C01807=1039.398,-71.584,-77.475,168.803,36.714,156.907
C01808=1039.391,-71.834,-77.463,168.801,36.714,156.907
C01809=1039.386,-72.084,-77.451,168.798,36.713,156.907
C01810=1039.380,-72.333,-77.439,168.796,36.713,156.907
C01811=1039.374,-72.584,-77.428,168.793,36.713,156.907
C01812=1039.368,-72.833,-77.417,168.791,36.713,156.907
C01813=1039.361,-73.083,-77.405,168.789,36.713,156.907
C01814=1039.356,-73.332,-77.394,168.786,36.713,156.907
C01815=1039.349,-73.582,-77.382,168.784,36.713,156.907
C01816=1039.344,-73.832,-77.371,168.781,36.713,156.907
C01817=1039.337,-74.082,-77.360,168.779,36.713,156.907
C01818=1039.331,-74.331,-77.348,168.776,36.713,156.907
C01819=1039.325,-74.581,-77.337,168.774,36.713,156.907
C01820=1039.319,-74.831,-77.325,168.772,36.713,156.907
C01821=1039.313,-75.080,-77.314,168.769,36.713,156.907
C01822=1039.306,-75.330,-77.303,168.767,36.713,156.907
C01823=1039.301,-75.580,-77.292,168.764,36.713,156.907
C01824=1039.294,-75.829,-77.280,168.762,36.713,156.907
C01825=1039.288,-76.079,-77.269,168.759,36.713,156.907
C01826=1039.282,-76.329,-77.258,168.757,36.713,156.907
C01827=1039.276,-76.578,-77.246,168.754,36.713,156.907
C01828=1039.269,-76.828,-77.235,168.752,36.714,156.907
C01829=1039.264,-77.077,-77.224,168.749,36.714,156.907
C01830=1039.257,-77.328,-77.213,168.747,36.714,156.907
C01831=1039.251,-77.576,-77.201,168.745,36.714,156.907
C01832=1039.244,-77.826,-77.190,168.742,36.714,156.907
C01833=1039.238,-78.076,-77.180,168.740,36.714,156.907
C01834=1039.232,-78.326,-77.168,168.737,36.714,156.907
C01835=1039.226,-78.575,-77.157,168.735,36.714,156.907
C01836=1039.220,-78.825,-77.146,168.732,36.714,156.907
C01837=1039.214,-79.075,-77.135,168.730,36.714,156.907
C01838=1039.208,-79.325,-77.123,168.727,36.714,156.907
C01839=1039.202,-79.574,-77.113,168.725,36.714,156.907
C01840=1039.196,-79.824,-77.101,168.722,36.714,156.907
C01841=1039.190,-80.074,-77.090,168.720,36.714,156.907
C01842=1039.182,-80.323,-77.079,168.717,36.714,156.907
C01843=1039.177,-80.573,-77.068,168.715,36.714,156.907
C01844=1039.170,-80.823,-77.057,168.712,36.714,156.907
C01845=1039.164,-81.072,-77.047,168.710,36.714,156.907
C01846=1039.158,-81.321,-77.036,168.707,36.715,156.907
C01847=1039.152,-81.572,-77.025,168.705,36.715,156.907
C01848=1039.145,-81.821,-77.014,168.702,36.715,156.907
C01849=1039.139,-82.071,-77.003,168.700,36.715,156.907
C01850=1039.133,-82.321,-76.992,168.697,36.716,156.908
C01851=1039.126,-82.570,-76.981,168.695,36.716,156.908
C01852=1039.120,-82.820,-76.971,168.692,36.716,156.908
C01853=1039.114,-83.070,-76.959,168.690,36.716,156.908
C01854=1039.108,-83.319,-76.949,168.687,36.716,156.908
C01855=1039.101,-83.605,-76.936,168.684,36.716,156.908
C01856=1039.094,-83.889,-76.924,168.682,36.717,156.908
C01857=1039.087,-84.174,-76.911,168.679,36.717,156.908
C01858=1039.080,-84.459,-76.899,168.676,36.717,156.908
C01859=1039.073,-84.709,-76.889,168.673,36.717,156.908
C01860=1039.067,-84.958,-76.878,168.672,36.718,156.908
C01861=1039.061,-85.209,-76.867,168.669,36.718,156.908
C01862=1039.054,-85.458,-76.856,168.667,36.718,156.908
C01863=1039.049,-85.707,-76.845,168.664,36.718,156.908
C01864=1039.042,-85.957,-76.834,168.662,36.719,156.908
C01865=1039.036,-86.207,-76.825,168.659,36.719,156.908
C01866=1039.030,-86.457,-76.814,168.657,36.719,156.908
C01867=1039.024,-86.707,-76.802,168.654,36.719,156.908
C01868=1039.018,-86.956,-76.792,168.652,36.719,156.908
C01869=1039.012,-87.206,-76.781,168.649,36.719,156.908
C01870=1039.005,-87.456,-76.770,168.647,36.719,156.908
C01871=1038.999,-87.705,-76.760,168.644,36.720,156.908
C01872=1038.993,-87.954,-76.749,168.642,36.720,156.908
C01873=1038.986,-88.205,-76.739,168.639,36.720,156.908
C01874=1038.981,-88.454,-76.728,168.637,36.721,156.908
C01875=1038.975,-88.704,-76.717,168.634,36.721,156.908
C01876=1038.968,-88.954,-76.707,168.631,36.721,156.908
C01877=1038.962,-89.203,-76.696,168.629,36.721,156.908
C01878=1038.957,-89.453,-76.685,168.626,36.721,156.908
C01879=1038.950,-89.703,-76.675,168.624,36.721,156.908
C01880=1038.944,-89.953,-76.664,168.621,36.722,156.908
C01881=1038.937,-90.202,-76.654,168.619,36.722,156.908
C01882=1038.932,-90.451,-76.643,168.616,36.722,156.908
C01883=1038.926,-90.702,-76.632,168.614,36.723,156.909
C01884=1038.919,-90.951,-76.622,168.611,36.723,156.909
C01885=1038.913,-91.201,-76.611,168.609,36.723,156.909
C01886=1038.907,-91.450,-76.601,168.606,36.723,156.909
C01887=1038.902,-91.700,-76.591,168.604,36.723,156.909
C01888=1038.895,-91.950,-76.579,168.601,36.724,156.909
C01889=1038.889,-92.200,-76.569,168.599,36.724,156.909
C01890=1038.883,-92.450,-76.559,168.596,36.724,156.909
C01891=1038.877,-92.699,-76.549,168.593,36.725,156.909
C01892=1038.870,-92.949,-76.537,168.591,36.725,156.909
C01893=1038.864,-93.199,-76.528,168.588,36.725,156.909
C01894=1038.859,-93.448,-76.517,168.586,36.726,156.909
C01895=1038.853,-93.698,-76.506,168.583,36.726,156.909
C01896=1038.847,-93.948,-76.497,168.581,36.726,156.909
C01897=1038.841,-94.197,-76.486,168.578,36.726,156.909
C01898=1038.834,-94.447,-76.475,168.576,36.726,156.909
C01899=1038.828,-94.697,-76.465,168.573,36.727,156.909
C01900=1038.823,-94.947,-76.454,168.571,36.727,156.909
C01901=1038.816,-95.196,-76.444,168.568,36.727,156.909
C01902=1038.811,-95.446,-76.434,168.566,36.728,156.909
C01903=1038.804,-95.695,-76.423,168.563,36.728,156.909
C01904=1038.799,-95.945,-76.413,168.561,36.728,156.909
C01905=1038.792,-96.195,-76.402,168.559,36.728,156.909
C01906=1038.786,-96.445,-76.392,168.556,36.728,156.909
C01907=1038.780,-96.694,-76.382,168.554,36.729,156.909
C01908=1038.774,-96.944,-76.372,168.551,36.729,156.909
C01909=1038.769,-97.194,-76.361,168.549,36.730,156.910
C01910=1038.762,-97.443,-76.351,168.546,36.730,156.910
C01911=1038.756,-97.693,-76.341,168.544,36.730,156.910
C01912=1038.751,-97.943,-76.331,168.541,36.730,156.910
C01913=1038.744,-98.193,-76.320,168.538,36.731,156.910
C01914=1038.737,-98.443,-76.311,168.536,36.731,156.910
C01915=1038.732,-98.692,-76.300,168.533,36.732,156.910
C01916=1038.725,-98.942,-76.290,168.531,36.732,156.910
C01917=1038.719,-99.191,-76.280,168.528,36.732,156.910
C01918=1038.714,-99.441,-76.270,168.525,36.733,156.910
C01919=1038.706,-99.729,-76.259,168.522,36.734,156.910
C01920=1038.699,-100.015,-76.247,168.519,36.734,156.910
C01921=1038.692,-100.303,-76.235,168.517,36.734,156.910
C01922=1038.685,-100.590,-76.224,168.514,36.735,156.910
C01923=1038.679,-100.840,-76.214,168.511,36.735,156.910
C01924=1038.673,-101.089,-76.203,168.508,36.736,156.911
C01925=1038.667,-101.339,-76.194,168.506,36.737,156.911
C01926=1038.660,-101.589,-76.184,168.503,36.737,156.911
C01927=1038.655,-101.839,-76.173,168.501,36.737,156.911
C01928=1038.649,-102.088,-76.164,168.498,36.737,156.911
C01929=1038.642,-102.338,-76.154,168.495,36.738,156.911
C01930=1038.636,-102.587,-76.144,168.494,36.739,156.911
C01931=1038.630,-102.837,-76.134,168.491,36.739,156.911
C01932=1038.624,-103.087,-76.124,168.489,36.739,156.911
C01933=1038.618,-103.336,-76.114,168.486,36.740,156.911
C01934=1038.612,-103.587,-76.104,168.483,36.740,156.911
C01935=1038.606,-103.836,-76.094,168.481,36.741,156.911
C01936=1038.600,-104.086,-76.084,168.478,36.741,156.911
C01937=1038.594,-104.335,-76.074,168.476,36.741,156.911
C01938=1038.588,-104.585,-76.064,168.473,36.742,156.911
C01939=1038.582,-104.835,-76.054,168.470,36.743,156.912
C01940=1038.576,-105.085,-76.045,168.468,36.743,156.912
C01941=1038.570,-105.335,-76.035,168.465,36.743,156.912
C01942=1038.564,-105.584,-76.024,168.463,36.744,156.912
C01943=1038.558,-105.834,-76.015,168.460,36.745,156.912
C01944=1038.552,-106.084,-76.005,168.457,36.745,156.912
C01945=1038.545,-106.334,-75.996,168.455,36.745,156.912
C01946=1038.539,-106.583,-75.986,168.452,36.746,156.912
C01947=1038.533,-106.833,-75.975,168.449,36.747,156.912
C01948=1038.527,-107.083,-75.966,168.447,36.747,156.912
///RCONF 1,0,0,0,1,0,0,0,0,0,0,0,0,0,0,0,0,0,0,0,0,0,0,0
C01949=1038.521,-107.333,-75.956,168.444,36.747,156.912
C01950=1038.515,-107.582,-75.947,168.442,36.748,156.912
C01951=1038.509,-107.832,-75.937,168.440,36.749,156.913
C01952=1038.503,-108.082,-75.927,168.437,36.749,156.913
C01953=1038.496,-108.332,-75.918,168.435,36.749,156.913
C01954=1038.490,-108.582,-75.908,168.432,36.750,156.913
C01955=1038.484,-108.831,-75.899,168.429,36.751,156.913
C01956=1038.479,-109.081,-75.889,168.427,36.751,156.913
C01957=1038.473,-109.331,-75.879,168.424,36.752,156.913
C01958=1038.467,-109.580,-75.870,168.422,36.753,156.913
C01959=1038.461,-109.830,-75.860,168.419,36.753,156.913
C01960=1038.454,-110.079,-75.850,168.416,36.754,156.913
C01961=1038.448,-110.329,-75.840,168.414,36.754,156.913
C01962=1038.442,-110.579,-75.831,168.411,36.755,156.914
C01963=1038.436,-110.829,-75.821,168.408,36.756,156.914
C01964=1038.430,-111.079,-75.812,168.406,36.756,156.914
C01965=1038.424,-111.329,-75.803,168.403,36.757,156.914
C01966=1038.418,-111.579,-75.793,168.400,36.757,156.914
C01967=1038.412,-111.828,-75.784,168.398,36.758,156.914
C01968=1038.406,-112.078,-75.774,168.395,36.758,156.914
C01969=1038.400,-112.327,-75.765,168.393,36.759,156.914
C01970=1038.393,-112.577,-75.755,168.391,36.760,156.914
C01971=1038.387,-112.827,-75.746,168.388,36.760,156.914
C01972=1038.381,-113.077,-75.736,168.386,36.761,156.914
C01973=1038.376,-113.326,-75.727,168.383,36.762,156.915
C01974=1038.369,-113.576,-75.717,168.380,36.762,156.915
C01975=1038.363,-113.826,-75.708,168.378,36.762,156.915
C01976=1038.358,-114.076,-75.698,168.375,36.763,156.915
C01977=1038.352,-114.325,-75.688,168.372,36.764,156.915
C01978=1038.345,-114.576,-75.680,168.370,36.764,156.915
C01979=1038.339,-114.825,-75.671,168.367,36.765,156.915
C01980=1038.333,-115.074,-75.661,168.364,36.766,156.915
C01981=1038.327,-115.324,-75.652,168.362,36.766,156.915
C01982=1038.321,-115.574,-75.642,168.359,36.767,156.915
C01983=1038.314,-115.861,-75.631,168.356,36.768,156.916
C01984=1038.307,-116.147,-75.621,168.354,36.769,156.916
C01985=1038.301,-116.433,-75.610,168.351,36.770,156.916
C01986=1038.294,-116.719,-75.599,168.348,36.770,156.916
C01987=1038.288,-116.969,-75.590,168.345,36.771,156.916
C01988=1038.282,-117.219,-75.580,168.342,36.772,156.916
C01989=1038.275,-117.469,-75.572,168.340,36.772,156.916
C01990=1038.269,-117.718,-75.563,168.337,36.773,156.916
C01991=1038.263,-117.968,-75.553,168.334,36.774,156.917
C01992=1038.257,-118.218,-75.544,168.332,36.774,156.917
C01993=1038.251,-118.468,-75.535,168.329,36.775,156.917
C01994=1038.246,-118.717,-75.526,168.326,36.776,156.917
C01995=1038.239,-118.967,-75.516,168.324,36.777,156.917
C01996=1038.233,-119.217,-75.508,168.321,36.777,156.917
C01997=1038.227,-119.467,-75.498,168.319,36.779,156.917
C01998=1038.221,-119.716,-75.489,168.317,36.779,156.917
C01999=1038.215,-119.967,-75.480,168.314,36.780,156.917
C02000=1038.209,-120.216,-75.471,168.311,36.781,156.918
C02001=1038.203,-120.465,-75.461,168.309,36.781,156.918
C02002=1038.197,-120.716,-75.453,168.306,36.782,156.918
C02003=1038.191,-120.965,-75.444,168.303,36.783,156.918
C02004=1038.185,-121.216,-75.435,168.301,36.783,156.918
C02005=1038.179,-121.465,-75.426,168.298,36.784,156.918
C02006=1038.173,-121.715,-75.416,168.295,36.785,156.918
C02007=1038.167,-121.965,-75.407,168.293,36.786,156.918
C02008=1038.161,-122.214,-75.399,168.290,36.787,156.919
C02009=1038.155,-122.464,-75.390,168.287,36.787,156.919
C02010=1038.149,-122.714,-75.380,168.286,36.788,156.919
C02011=1038.143,-122.963,-75.371,168.283,36.789,156.919
C02012=1038.137,-123.213,-75.363,168.280,36.789,156.919
C02013=1038.131,-123.463,-75.353,168.277,36.791,156.919
C02014=1038.125,-123.713,-75.345,168.275,36.791,156.919
C02015=1038.119,-123.963,-75.335,168.272,36.792,156.919
C02016=1038.114,-124.212,-75.327,168.269,36.793,156.920
C02017=1038.107,-124.462,-75.318,168.267,36.793,156.920
C02018=1038.101,-124.712,-75.309,168.264,36.794,156.920
C02019=1038.095,-124.961,-75.300,168.261,36.795,156.920
C02020=1038.089,-125.211,-75.291,168.259,36.796,156.920
C02021=1038.083,-125.461,-75.282,168.256,36.797,156.920
C02022=1038.077,-125.711,-75.273,168.254,36.798,156.920
C02023=1038.071,-125.961,-75.265,168.251,36.799,156.920
C02024=1038.065,-126.210,-75.256,168.249,36.800,156.921
C02025=1038.059,-126.461,-75.247,168.246,36.800,156.921
C02026=1038.053,-126.710,-75.238,168.243,36.802,156.921
C02027=1038.047,-126.960,-75.230,168.241,36.802,156.921
C02028=1038.041,-127.210,-75.221,168.238,36.803,156.921
C02029=1038.035,-127.459,-75.212,168.235,36.804,156.921
C02030=1038.029,-127.709,-75.203,168.233,36.805,156.921
C02031=1038.024,-127.958,-75.194,168.230,36.806,156.922
C02032=1038.019,-128.208,-75.184,168.227,36.806,156.922
C02033=1038.014,-128.458,-75.175,168.225,36.806,156.922
C02034=1038.011,-128.708,-75.164,168.223,36.805,156.921
C02035=1038.008,-128.958,-75.153,168.221,36.804,156.921
C02036=1038.007,-129.208,-75.140,168.219,36.802,156.921
C02037=1038.005,-129.458,-75.128,168.217,36.800,156.921
C02038=1038.005,-129.707,-75.115,168.215,36.798,156.920
C02039=1038.005,-129.957,-75.101,168.213,36.794,156.920
C02040=1038.006,-130.208,-75.086,168.212,36.791,156.919
C02041=1038.009,-130.458,-75.071,168.210,36.787,156.918
C02042=1038.012,-130.707,-75.057,168.209,36.783,156.918
C02043=1038.015,-130.959,-75.041,168.207,36.779,156.917
C02044=1038.019,-131.208,-75.024,168.207,36.773,156.916
C02045=1038.024,-131.459,-75.006,168.205,36.767,156.915
C02046=1038.030,-131.708,-74.989,168.205,36.761,156.914
C02047=1037.689,-131.732,-75.257,168.156,36.967,156.948
C02048=1037.683,-131.483,-75.275,168.158,36.973,156.949
C02049=1037.679,-131.233,-75.293,168.158,36.978,156.950
C02050=1037.674,-130.983,-75.309,168.160,36.984,156.951
C02051=1037.671,-130.732,-75.326,168.161,36.988,156.952
C02052=1037.668,-130.483,-75.340,168.162,36.993,156.953
C02053=1037.666,-130.232,-75.356,168.164,36.997,156.954
C02054=1037.665,-129.982,-75.370,168.166,37.000,156.954
C02055=1037.664,-129.732,-75.384,168.167,37.003,156.955
C02056=1037.665,-129.482,-75.397,168.169,37.006,156.955
C02057=1037.665,-129.232,-75.410,168.171,37.007,156.955
C02058=1037.668,-128.983,-75.421,168.173,37.009,156.956
C02059=1037.670,-128.733,-75.433,168.175,37.010,156.956
C02060=1037.674,-128.483,-75.444,168.178,37.011,156.956
C02061=1037.677,-128.232,-75.454,168.180,37.011,156.956
C02062=1037.682,-127.983,-75.464,168.182,37.011,156.956
C02063=1037.688,-127.734,-75.473,168.185,37.010,156.956
C02064=1037.694,-127.484,-75.481,168.188,37.009,156.956
C02065=1037.700,-127.234,-75.490,168.190,37.009,156.956
C02066=1037.706,-126.984,-75.499,168.193,37.007,156.955
C02067=1037.712,-126.735,-75.507,168.196,37.007,156.955
C02068=1037.718,-126.485,-75.516,168.199,37.006,156.955
C02069=1037.724,-126.234,-75.525,168.200,37.004,156.955
C02070=1037.730,-125.986,-75.534,168.203,37.004,156.955
C02071=1037.736,-125.735,-75.543,168.206,37.003,156.955
C02072=1037.741,-125.486,-75.551,168.209,37.002,156.955
C02073=1037.748,-125.236,-75.560,168.211,37.001,156.954
C02074=1037.754,-124.986,-75.569,168.214,37.000,156.954
C02075=1037.760,-124.737,-75.578,168.217,37.000,156.954
C02076=1037.766,-124.486,-75.587,168.219,36.998,156.954
C02077=1037.772,-124.237,-75.596,168.222,36.998,156.954
C02078=1037.778,-123.987,-75.605,168.225,36.997,156.954
C02079=1037.784,-123.737,-75.614,168.228,36.996,156.954
C02080=1037.790,-123.488,-75.622,168.229,36.995,156.953
C02081=1037.796,-123.238,-75.632,168.232,36.994,156.953
C02082=1037.802,-122.987,-75.640,168.235,36.993,156.953
C02083=1037.808,-122.738,-75.650,168.237,36.993,156.953
C02084=1037.814,-122.488,-75.658,168.240,36.992,156.953
C02085=1037.820,-122.238,-75.668,168.243,36.991,156.953
C02086=1037.826,-121.989,-75.676,168.245,36.990,156.953
C02087=1037.832,-121.739,-75.686,168.248,36.989,156.953
C02088=1037.838,-121.489,-75.695,168.251,36.989,156.953
C02089=1037.844,-121.240,-75.703,168.254,36.988,156.952
C02090=1037.850,-120.990,-75.713,168.256,36.987,156.952
C02091=1037.856,-120.740,-75.721,168.258,36.986,156.952
C02092=1037.861,-120.490,-75.731,168.261,36.985,156.952
C02093=1037.868,-120.241,-75.740,168.263,36.984,156.952
C02094=1037.874,-119.990,-75.749,168.266,36.984,156.952
C02095=1037.880,-119.741,-75.758,168.269,36.983,156.952
C02096=1037.886,-119.492,-75.767,168.271,36.982,156.952
C02097=1037.892,-119.241,-75.776,168.274,36.982,156.952
C02098=1037.898,-118.991,-75.786,168.277,36.980,156.951
C02099=1037.904,-118.742,-75.795,168.280,36.980,156.951
C02100=1037.909,-118.492,-75.804,168.282,36.979,156.951
C02101=1037.916,-118.242,-75.813,168.285,36.978,156.951
C02102=1037.923,-117.993,-75.822,168.288,36.978,156.951
C02103=1037.928,-117.744,-75.831,168.290,36.977,156.951
C02104=1037.934,-117.493,-75.840,168.292,36.976,156.951
C02105=1037.940,-117.243,-75.850,168.295,36.975,156.951
C02106=1037.946,-116.994,-75.859,168.297,36.975,156.950
C02107=1037.952,-116.744,-75.868,168.300,36.974,156.950
C02108=1037.959,-116.458,-75.879,168.303,36.973,156.950
C02109=1037.966,-116.172,-75.890,168.306,36.972,156.950
C02110=1037.973,-115.885,-75.901,168.309,36.971,156.950
C02111=1037.980,-115.599,-75.911,168.312,36.971,156.950
C02112=1037.986,-115.349,-75.920,168.315,36.970,156.950
C02113=1037.992,-115.099,-75.929,168.318,36.969,156.950
C02114=1037.998,-114.849,-75.939,168.320,36.969,156.950
C02115=1038.004,-114.600,-75.948,168.323,36.968,156.949
C02116=1038.010,-114.350,-75.958,168.326,36.967,156.949
C02117=1038.016,-114.100,-75.967,168.327,36.967,156.949
C02118=1038.022,-113.851,-75.976,168.330,36.966,156.949
C02119=1038.028,-113.600,-75.985,168.333,36.965,156.949
C02120=1038.034,-113.351,-75.995,168.335,36.964,156.949
C02121=1038.040,-113.101,-76.004,168.338,36.964,156.949
C02122=1038.046,-112.851,-76.014,168.341,36.963,156.949
C02123=1038.052,-112.601,-76.024,168.343,36.962,156.949
C02124=1038.058,-112.352,-76.033,168.346,36.962,156.948
C02125=1038.064,-112.102,-76.042,168.349,36.961,156.948
C02126=1038.070,-111.853,-76.052,168.351,36.960,156.948
C02127=1038.077,-111.603,-76.061,168.354,36.960,156.948
C02128=1038.083,-111.353,-76.071,168.357,36.959,156.948
C02129=1038.089,-111.103,-76.081,168.359,36.958,156.948
C02130=1038.095,-110.853,-76.090,168.362,36.958,156.948
C02131=1038.101,-110.604,-76.100,168.365,36.957,156.948
C02132=1038.106,-110.354,-76.110,168.366,36.957,156.948
C02133=1038.112,-110.104,-76.119,168.369,36.956,156.948
C02134=1038.118,-109.855,-76.129,168.372,36.955,156.948
C02135=1038.125,-109.605,-76.138,168.374,36.955,156.947
C02136=1038.131,-109.355,-76.148,168.377,36.954,156.947
C02137=1038.137,-109.105,-76.157,168.380,36.953,156.947
C02138=1038.143,-108.855,-76.167,168.382,36.953,156.947
C02139=1038.149,-108.606,-76.176,168.385,36.952,156.947
C02140=1038.155,-108.356,-76.186,168.388,36.952,156.947
C02141=1038.162,-108.106,-76.196,168.390,36.951,156.947
C02142=1038.168,-107.856,-76.205,168.393,36.951,156.947
C02143=1038.174,-107.606,-76.215,168.396,36.950,156.947
C02144=1038.180,-107.357,-76.224,168.398,36.949,156.947
C02145=1038.185,-107.107,-76.234,168.401,36.949,156.947
C02146=1038.191,-106.858,-76.244,168.403,36.948,156.947
C02147=1038.198,-106.608,-76.254,168.406,36.948,156.946
C02148=1038.204,-106.358,-76.264,168.409,36.947,156.946
C02149=1038.210,-106.109,-76.273,168.410,36.946,156.946
C02150=1038.215,-105.858,-76.283,168.413,36.946,156.946
C02151=1038.222,-105.609,-76.293,168.416,36.946,156.946
C02152=1038.228,-105.360,-76.303,168.418,36.945,156.946
///RCONF 1,0,0,0,0,0,0,0,0,0,0,0,0,0,0,0,0,0,0,0,0,0,0,0
C02153=1038.234,-105.110,-76.313,168.421,36.944,156.946
C02154=1038.240,-104.860,-76.323,168.423,36.944,156.946
C02155=1038.246,-104.610,-76.332,168.426,36.944,156.946
C02156=1038.252,-104.360,-76.342,168.429,36.943,156.946
C02157=1038.258,-104.111,-76.352,168.431,36.942,156.946
C02158=1038.264,-103.861,-76.362,168.434,36.942,156.946
C02159=1038.270,-103.611,-76.372,168.437,36.942,156.945
C02160=1038.276,-103.361,-76.382,168.439,36.941,156.945
C02161=1038.283,-103.112,-76.392,168.442,36.940,156.945
C02162=1038.288,-102.862,-76.402,168.444,36.940,156.945
C02163=1038.294,-102.612,-76.412,168.447,36.939,156.945
C02164=1038.301,-102.363,-76.422,168.450,36.939,156.945
C02165=1038.307,-102.113,-76.431,168.452,36.939,156.945
C02166=1038.312,-101.863,-76.442,168.455,36.938,156.945
C02167=1038.319,-101.614,-76.452,168.457,36.937,156.945
C02168=1038.325,-101.364,-76.461,168.460,36.937,156.945
C02169=1038.331,-101.114,-76.472,168.462,36.937,156.945
C02170=1038.338,-100.864,-76.482,168.464,36.936,156.945
C02171=1038.344,-100.614,-76.492,168.467,36.936,156.945
C02172=1038.350,-100.327,-76.503,168.470,36.935,156.945
C02173=1038.357,-100.040,-76.515,168.473,36.935,156.944
C02174=1038.365,-99.753,-76.526,168.476,36.934,156.944
C02175=1038.371,-99.466,-76.538,168.479,36.933,156.944
C02176=1038.377,-99.216,-76.548,168.482,36.933,156.944
C02177=1038.384,-98.967,-76.558,168.484,36.932,156.944
C02178=1038.389,-98.717,-76.568,168.487,36.932,156.944
C02179=1038.396,-98.466,-76.578,168.489,36.932,156.944
C02180=1038.403,-98.217,-76.589,168.492,36.931,156.944
C02181=1038.409,-97.967,-76.598,168.495,36.931,156.944
C02182=1038.414,-97.718,-76.609,168.497,36.930,156.944
C02183=1038.421,-97.468,-76.619,168.500,36.930,156.944
C02184=1038.426,-97.218,-76.629,168.502,36.930,156.944
C02185=1038.433,-96.968,-76.639,168.505,36.929,156.944
C02186=1038.438,-96.719,-76.650,168.507,36.929,156.944
C02187=1038.444,-96.469,-76.659,168.510,36.928,156.944
C02188=1038.451,-96.219,-76.671,168.513,36.928,156.944
C02189=1038.457,-95.970,-76.681,168.515,36.928,156.944
C02190=1038.463,-95.720,-76.691,168.518,36.927,156.943
C02191=1038.468,-95.470,-76.702,168.520,36.927,156.943
C02192=1038.475,-95.220,-76.712,168.523,36.927,156.943
C02193=1038.480,-94.971,-76.722,168.525,36.927,156.943
C02194=1038.487,-94.721,-76.732,168.527,36.926,156.943
C02195=1038.493,-94.471,-76.743,168.530,36.926,156.943
C02196=1038.499,-94.222,-76.754,168.532,36.925,156.943
C02197=1038.505,-93.972,-76.764,168.535,36.925,156.943
C02198=1038.511,-93.722,-76.775,168.537,36.925,156.943
C02199=1038.517,-93.473,-76.785,168.540,36.925,156.943
C02200=1038.522,-93.223,-76.795,168.542,36.925,156.943
C02201=1038.530,-92.973,-76.806,168.545,36.924,156.943
C02202=1038.535,-92.724,-76.817,168.547,36.924,156.943
C02203=1038.541,-92.473,-76.827,168.550,36.923,156.943
C02204=1038.547,-92.224,-76.837,168.553,36.923,156.943
C02205=1038.553,-91.975,-76.848,168.555,36.923,156.943
C02206=1038.560,-91.724,-76.858,168.558,36.922,156.943
C02207=1038.565,-91.475,-76.869,168.560,36.922,156.943
C02208=1038.572,-91.226,-76.879,168.563,36.922,156.943
C02209=1038.578,-90.976,-76.890,168.565,36.922,156.943
C02210=1038.584,-90.725,-76.900,168.568,36.922,156.943
C02211=1038.590,-90.476,-76.911,168.570,36.921,156.943
C02212=1038.596,-90.227,-76.922,168.573,36.921,156.943
C02213=1038.602,-89.977,-76.932,168.576,36.920,156.943
C02214=1038.608,-89.727,-76.942,168.578,36.920,156.943
C02215=1038.614,-89.477,-76.953,168.581,36.920,156.943
C02216=1038.621,-89.228,-76.963,168.583,36.920,156.942
C02217=1038.626,-88.978,-76.974,168.586,36.919,156.942
C02218=1038.632,-88.728,-76.985,168.588,36.919,156.942
C02219=1038.639,-88.478,-76.995,168.591,36.919,156.942
C02220=1038.645,-88.229,-77.006,168.593,36.919,156.942
C02221=1038.652,-87.979,-77.017,168.596,36.918,156.942
C02222=1038.657,-87.730,-77.028,168.598,36.918,156.942
C02223=1038.663,-87.480,-77.038,168.601,36.918,156.942
C02224=1038.670,-87.230,-77.048,168.603,36.917,156.942
C02225=1038.676,-86.980,-77.059,168.606,36.917,156.942
C02226=1038.681,-86.731,-77.070,168.609,36.917,156.942
C02227=1038.688,-86.481,-77.081,168.611,36.917,156.942
C02228=1038.694,-86.231,-77.092,168.614,36.917,156.942
C02229=1038.700,-85.982,-77.103,168.616,36.917,156.942
C02230=1038.707,-85.732,-77.113,168.619,36.916,156.942
C02231=1038.713,-85.482,-77.124,168.621,36.916,156.942
C02232=1038.719,-85.233,-77.134,168.624,36.916,156.942
C02233=1038.726,-84.983,-77.146,168.625,36.915,156.942
C02234=1038.731,-84.734,-77.156,168.628,36.915,156.942
C02235=1038.738,-84.484,-77.166,168.630,36.915,156.942
C02236=1038.745,-84.199,-77.179,168.633,36.914,156.942
C02237=1038.752,-83.913,-77.192,168.636,36.914,156.942
C02238=1038.758,-83.629,-77.204,168.639,36.914,156.942
C02239=1038.766,-83.343,-77.216,168.642,36.914,156.942
C02240=1038.772,-83.094,-77.226,168.644,36.914,156.942
C02241=1038.779,-82.844,-77.238,168.647,36.913,156.942
C02242=1038.784,-82.594,-77.249,168.650,36.913,156.942
C02243=1038.791,-82.345,-77.259,168.652,36.913,156.942
C02244=1038.797,-82.095,-77.270,168.655,36.913,156.942
C02245=1038.804,-81.845,-77.281,168.657,36.912,156.941
C02246=1038.810,-81.596,-77.292,168.660,36.912,156.941
C02247=1038.816,-81.346,-77.303,168.662,36.912,156.941
C02248=1038.822,-81.096,-77.314,168.665,36.911,156.941
C02249=1038.829,-80.848,-77.325,168.667,36.911,156.941
C02250=1038.835,-80.597,-77.336,168.670,36.911,156.941
C02251=1038.841,-80.348,-77.347,168.672,36.911,156.941
C02252=1038.847,-80.098,-77.358,168.675,36.911,156.941
C02253=1038.854,-79.848,-77.368,168.677,36.911,156.941
C02254=1038.860,-79.598,-77.380,168.680,36.911,156.941
C02255=1038.866,-79.349,-77.391,168.682,36.911,156.941
C02256=1038.872,-79.099,-77.402,168.685,36.911,156.941
C02257=1038.878,-78.850,-77.413,168.687,36.910,156.941
C02258=1038.885,-78.600,-77.425,168.690,36.910,156.941
C02259=1038.890,-78.350,-77.435,168.692,36.910,156.941
C02260=1038.897,-78.100,-77.447,168.695,36.910,156.941
C02261=1038.902,-77.850,-77.458,168.697,36.910,156.941
C02262=1038.909,-77.601,-77.470,168.700,36.910,156.941
C02263=1038.915,-77.352,-77.480,168.702,36.910,156.941
C02264=1038.922,-77.101,-77.491,168.705,36.910,156.941
C02265=1038.928,-76.852,-77.502,168.707,36.910,156.941
C02266=1038.934,-76.602,-77.514,168.709,36.909,156.941
C02267=1038.940,-76.353,-77.525,168.712,36.909,156.941
C02268=1038.946,-76.103,-77.536,168.714,36.909,156.941
C02269=1038.952,-75.853,-77.547,168.717,36.909,156.941
C02270=1038.959,-75.604,-77.559,168.719,36.909,156.941
C02271=1038.964,-75.354,-77.570,168.722,36.909,156.941
C02272=1038.971,-75.104,-77.581,168.724,36.909,156.941
C02273=1038.977,-74.855,-77.593,168.727,36.909,156.941
C02274=1038.983,-74.605,-77.604,168.729,36.909,156.941
C02275=1038.989,-74.355,-77.615,168.732,36.909,156.941
C02276=1038.996,-74.106,-77.627,168.734,36.909,156.941
C02277=1039.002,-73.856,-77.638,168.737,36.909,156.941
C02278=1039.008,-73.606,-77.649,168.739,36.909,156.941
C02279=1039.014,-73.357,-77.661,168.741,36.909,156.941
C02280=1039.019,-73.107,-77.672,168.744,36.909,156.941
C02281=1039.026,-72.857,-77.684,168.746,36.909,156.941
C02282=1039.032,-72.608,-77.695,168.749,36.909,156.941
C02283=1039.038,-72.358,-77.707,168.751,36.909,156.941
C02284=1039.044,-72.109,-77.718,168.754,36.909,156.941
C02285=1039.050,-71.859,-77.730,168.756,36.909,156.941
C02286=1039.056,-71.609,-77.741,168.758,36.909,156.941
C02287=1039.062,-71.359,-77.753,168.761,36.909,156.941
C02288=1039.069,-71.109,-77.765,168.763,36.909,156.941
C02289=1039.074,-70.860,-77.776,168.766,36.909,156.941
C02290=1039.080,-70.610,-77.788,168.768,36.909,156.941
C02291=1039.086,-70.361,-77.800,168.770,36.909,156.941
C02292=1039.093,-70.111,-77.811,168.773,36.909,156.941
C02293=1039.099,-69.861,-77.823,168.775,36.910,156.942
C02294=1039.104,-69.612,-77.834,168.778,36.910,156.942
C02295=1039.111,-69.362,-77.846,168.780,36.910,156.942
C02296=1039.117,-69.113,-77.857,168.782,36.910,156.942
C02297=1039.123,-68.863,-77.869,168.785,36.910,156.942
C02298=1039.129,-68.613,-77.881,168.787,36.909,156.942
C02299=1039.135,-68.364,-77.892,168.790,36.909,156.942
C02300=1039.142,-68.080,-77.906,168.792,36.910,156.942
C02301=1039.149,-67.798,-77.919,168.795,36.910,156.942
C02302=1039.156,-67.515,-77.932,168.798,36.910,156.942
C02303=1039.163,-67.233,-77.946,168.801,36.910,156.942
C02304=1039.169,-66.983,-77.957,168.803,36.910,156.942
C02305=1039.175,-66.733,-77.969,168.805,36.910,156.942
C02306=1039.181,-66.484,-77.981,168.808,36.911,156.942
C02307=1039.188,-66.234,-77.992,168.810,36.911,156.942
C02308=1039.194,-65.984,-78.004,168.813,36.911,156.942
C02309=1039.200,-65.734,-78.017,168.815,36.910,156.942
C02310=1039.206,-65.485,-78.028,168.817,36.910,156.942
C02311=1039.212,-65.235,-78.040,168.820,36.910,156.942
C02312=1039.219,-64.986,-78.051,168.823,36.911,156.942
C02313=1039.224,-64.736,-78.063,168.826,36.911,156.942
C02314=1039.231,-64.486,-78.075,168.828,36.911,156.942
C02315=1039.237,-64.237,-78.087,168.830,36.911,156.942
C02316=1039.243,-63.987,-78.099,168.833,36.911,156.942
C02317=1039.249,-63.737,-78.110,168.835,36.911,156.942
C02318=1039.256,-63.488,-78.122,168.837,36.912,156.942
C02319=1039.262,-63.238,-78.134,168.840,36.912,156.942
C02320=1039.268,-62.988,-78.147,168.842,36.912,156.942
C02321=1039.274,-62.739,-78.158,168.845,36.911,156.942
C02322=1039.281,-62.489,-78.170,168.847,36.911,156.942
C02323=1039.287,-62.239,-78.182,168.849,36.912,156.942
C02324=1039.293,-61.990,-78.194,168.852,36.912,156.942
C02325=1039.299,-61.741,-78.206,168.854,36.912,156.942
C02326=1039.305,-61.490,-78.218,168.857,36.912,156.942
C02327=1039.312,-61.241,-78.230,168.859,36.912,156.942
C02328=1039.318,-60.991,-78.241,168.861,36.913,156.942
C02329=1039.325,-60.742,-78.253,168.864,36.913,156.942
C02330=1039.330,-60.493,-78.266,168.866,36.913,156.942
C02331=1039.337,-60.243,-78.278,168.868,36.913,156.942
C02332=1039.343,-59.993,-78.289,168.871,36.913,156.942
C02333=1039.349,-59.743,-78.301,168.873,36.913,156.943
C02334=1039.356,-59.493,-78.313,168.876,36.913,156.943
C02335=1039.362,-59.244,-78.325,168.878,36.913,156.943
C02336=1039.368,-58.995,-78.337,168.880,36.913,156.943
C02337=1039.374,-58.745,-78.349,168.883,36.914,156.943
C02338=1039.381,-58.495,-78.361,168.885,36.914,156.943
C02339=1039.387,-58.246,-78.374,168.887,36.914,156.943
C02340=1039.393,-57.996,-78.386,168.890,36.914,156.943
C02341=1039.400,-57.746,-78.398,168.892,36.914,156.943
C02342=1039.406,-57.496,-78.410,168.895,36.914,156.943
C02343=1039.412,-57.246,-78.422,168.897,36.914,156.943
C02344=1039.418,-56.997,-78.433,168.899,36.914,156.943
C02345=1039.424,-56.748,-78.446,168.902,36.914,156.943
C02346=1039.431,-56.498,-78.458,168.904,36.915,156.943
C02347=1039.438,-56.248,-78.470,168.906,36.915,156.943
C02348=1039.444,-55.999,-78.482,168.909,36.915,156.943
C02349=1039.450,-55.749,-78.494,168.911,36.915,156.943
C02350=1039.457,-55.499,-78.506,168.913,36.915,156.943
C02351=1039.463,-55.249,-78.519,168.916,36.915,156.943
C02352=1039.469,-55.000,-78.531,168.918,36.915,156.943
C02353=1039.476,-54.751,-78.544,168.921,36.915,156.943
C02354=1039.482,-54.501,-78.556,168.923,36.915,156.943
C02355=1039.489,-54.252,-78.568,168.925,36.916,156.943
C02356=1039.495,-54.002,-78.580,168.928,36.916,156.943
C02357=1039.501,-53.753,-78.592,168.930,36.916,156.943
C02358=1039.507,-53.503,-78.604,168.932,36.916,156.943
C02359=1039.513,-53.253,-78.617,168.935,36.916,156.943
C02360=1039.520,-53.004,-78.629,168.937,36.916,156.943
C02361=1039.527,-52.754,-78.640,168.939,36.916,156.943
C02362=1039.533,-52.504,-78.653,168.943,36.916,156.943
C02363=1039.539,-52.255,-78.665,168.945,36.917,156.944
C02364=1039.547,-51.973,-78.679,168.948,36.917,156.944
C02365=1039.554,-51.691,-78.693,168.950,36.917,156.944
C02366=1039.561,-51.410,-78.708,168.953,36.917,156.944
C02367=1039.569,-51.128,-78.721,168.956,36.917,156.944
C02368=1039.575,-50.879,-78.734,168.958,36.917,156.944
C02369=1039.582,-50.629,-78.746,168.960,36.917,156.944
C02370=1039.588,-50.379,-78.758,168.963,36.918,156.944
C02371=1039.593,-50.129,-78.771,168.965,36.918,156.944
C02372=1039.600,-49.880,-78.783,168.967,36.919,156.944
C02373=1039.606,-49.631,-78.796,168.969,36.919,156.944
C02374=1039.612,-49.381,-78.809,168.972,36.919,156.944
C02375=1039.619,-49.131,-78.821,168.974,36.919,156.944
C02376=1039.625,-48.882,-78.834,168.976,36.920,156.944
C02377=1039.631,-48.632,-78.847,168.979,36.920,156.944
C02378=1039.637,-48.382,-78.859,168.981,36.920,156.944
C02379=1039.644,-48.133,-78.871,168.983,36.920,156.944
C02380=1039.650,-47.883,-78.884,168.985,36.921,156.945
C02381=1039.656,-47.633,-78.897,168.988,36.921,156.945
C02382=1039.662,-47.384,-78.910,168.990,36.922,156.945
C02383=1039.669,-47.135,-78.922,168.992,36.922,156.945
C02384=1039.674,-46.885,-78.935,168.995,36.922,156.945
C02385=1039.681,-46.635,-78.948,168.997,36.922,156.945
C02386=1039.687,-46.386,-78.961,168.999,36.923,156.945
C02387=1039.693,-46.136,-78.972,169.001,36.923,156.945
C02388=1039.699,-45.887,-78.986,169.005,36.923,156.945
C02389=1039.705,-45.637,-78.998,169.007,36.924,156.945
C02390=1039.712,-45.388,-79.012,169.009,36.924,156.945
C02391=1039.718,-45.138,-79.024,169.011,36.925,156.945
C02392=1039.724,-44.888,-79.036,169.014,36.925,156.945
C02393=1039.730,-44.639,-79.049,169.016,36.925,156.945
C02394=1039.736,-44.389,-79.062,169.018,36.925,156.945
C02395=1039.743,-44.140,-79.075,169.020,36.926,156.946
C02396=1039.749,-43.890,-79.087,169.023,36.926,156.946
C02397=1039.756,-43.640,-79.101,169.025,36.926,156.946
C02398=1039.762,-43.390,-79.113,169.027,36.926,156.946
C02399=1039.769,-43.141,-79.126,169.030,36.927,156.946
C02400=1039.775,-42.891,-79.139,169.032,36.927,156.946
C02401=1039.781,-42.642,-79.152,169.034,36.928,156.946
C02402=1039.787,-42.392,-79.164,169.036,36.928,156.946
C02403=1039.793,-42.143,-79.178,169.039,36.928,156.946
C02404=1039.800,-41.894,-79.190,169.041,36.928,156.946
C02405=1039.806,-41.644,-79.203,169.043,36.929,156.946
C02406=1039.812,-41.394,-79.216,169.045,36.929,156.946
C02407=1039.819,-41.144,-79.229,169.048,36.929,156.946
C02408=1039.825,-40.895,-79.241,169.050,36.930,156.946
C02409=1039.831,-40.646,-79.254,169.052,36.930,156.946
C02410=1039.838,-40.396,-79.268,169.055,36.931,156.947
C02411=1039.844,-40.146,-79.280,169.058,36.931,156.947
C02412=1039.850,-39.896,-79.294,169.060,36.931,156.947
C02413=1039.857,-39.647,-79.306,169.062,36.931,156.947
C02414=1039.863,-39.398,-79.319,169.064,36.932,156.947
C02415=1039.869,-39.148,-79.332,169.067,36.932,156.947
C02416=1039.876,-38.898,-79.345,169.069,36.932,156.947
C02417=1039.882,-38.648,-79.358,169.071,36.933,156.947
C02418=1039.888,-38.399,-79.372,169.073,36.933,156.947
C02419=1039.894,-38.149,-79.384,169.075,36.934,156.947
C02420=1039.901,-37.900,-79.398,169.078,36.934,156.947
C02421=1039.907,-37.650,-79.411,169.080,36.934,156.947
C02422=1039.913,-37.400,-79.424,169.082,36.935,156.947
C02423=1039.919,-37.151,-79.437,169.084,36.935,156.948
C02424=1039.926,-36.902,-79.450,169.086,36.936,156.948
C02425=1039.932,-36.652,-79.464,169.089,36.936,156.948
C02426=1039.938,-36.402,-79.476,169.091,36.937,156.948
C02427=1039.945,-36.153,-79.490,169.093,36.937,156.948
C02428=1039.951,-35.872,-79.505,169.096,36.938,156.948
C02429=1039.958,-35.591,-79.520,169.098,36.938,156.948
C02430=1039.966,-35.309,-79.534,169.101,36.939,156.948
C02431=1039.973,-35.028,-79.550,169.104,36.939,156.948
C02432=1039.979,-34.779,-79.563,169.106,36.940,156.948
C02433=1039.985,-34.530,-79.576,169.108,36.940,156.948
C02434=1039.991,-34.280,-79.589,169.111,36.940,156.949
C02435=1039.998,-34.030,-79.602,169.113,36.941,156.949
C02436=1040.004,-33.781,-79.616,169.115,36.941,156.949
C02437=1040.010,-33.531,-79.629,169.117,36.942,156.949
C02438=1040.016,-33.282,-79.642,169.119,36.942,156.949
C02439=1040.023,-33.032,-79.656,169.121,36.943,156.949
C02440=1040.029,-32.783,-79.669,169.124,36.943,156.949
C02441=1040.035,-32.533,-79.682,169.126,36.943,156.949
C02442=1040.041,-32.283,-79.696,169.128,36.944,156.949
C02443=1040.048,-32.033,-79.709,169.130,36.945,156.949
C02444=1040.054,-31.784,-79.722,169.132,36.945,156.949
C02445=1040.061,-31.534,-79.736,169.135,36.945,156.950
C02446=1040.067,-31.285,-79.749,169.138,36.946,156.950
C02447=1040.073,-31.036,-79.763,169.140,36.946,156.950
C02448=1040.079,-30.786,-79.776,169.142,36.946,156.950
C02449=1040.086,-30.536,-79.790,169.144,36.947,156.950
C02450=1040.092,-30.287,-79.803,169.146,36.948,156.950
C02451=1040.099,-30.038,-79.816,169.149,36.948,156.950
C02452=1040.105,-29.788,-79.830,169.151,36.948,156.950
C02453=1040.112,-29.539,-79.843,169.153,36.949,156.950
C02454=1040.118,-29.288,-79.857,169.155,36.950,156.950
C02455=1040.124,-29.039,-79.870,169.157,36.949,156.950
C02456=1040.130,-28.790,-79.884,169.159,36.950,156.951
C02457=1040.137,-28.540,-79.897,169.162,36.951,156.951
C02458=1040.143,-28.291,-79.911,169.164,36.951,156.951
C02459=1040.149,-28.041,-79.924,169.166,36.951,156.951
C02460=1040.156,-27.791,-79.938,169.168,36.952,156.951
C02461=1040.162,-27.542,-79.951,169.170,36.953,156.951
C02462=1040.169,-27.292,-79.964,169.172,36.953,156.951
C02463=1040.175,-27.043,-79.978,169.176,36.953,156.951
C02464=1040.181,-26.793,-79.992,169.178,36.954,156.951
C02465=1040.188,-26.543,-80.005,169.180,36.954,156.951
C02466=1040.193,-26.294,-80.019,169.182,36.955,156.952
C02467=1040.200,-26.044,-80.033,169.184,36.956,156.952
C02468=1040.206,-25.795,-80.046,169.186,36.956,156.952
C02469=1040.212,-25.545,-80.060,169.188,36.956,156.952
C02470=1040.219,-25.296,-80.074,169.191,36.957,156.952
C02471=1040.225,-25.046,-80.087,169.193,36.957,156.952
C02472=1040.231,-24.796,-80.102,169.195,36.958,156.952
C02473=1040.237,-24.547,-80.115,169.197,36.959,156.952
C02474=1040.243,-24.298,-80.128,169.199,36.959,156.952
C02475=1040.250,-24.047,-80.143,169.201,36.960,156.953
C02476=1040.256,-23.799,-80.156,169.204,36.961,156.953
C02477=1040.263,-23.549,-80.170,169.206,36.961,156.953
C02478=1040.268,-23.299,-80.184,169.208,36.961,156.953
C02479=1040.275,-23.049,-80.198,169.211,36.962,156.953
C02480=1040.281,-22.800,-80.212,169.213,36.962,156.953
C02481=1040.287,-22.551,-80.225,169.215,36.963,156.953
C02482=1040.294,-22.301,-80.239,169.217,36.964,156.953
C02483=1040.299,-22.051,-80.253,169.219,36.964,156.953
C02484=1040.307,-21.802,-80.267,169.221,36.965,156.953
C02485=1040.313,-21.553,-80.281,169.223,36.965,156.954
C02486=1040.319,-21.303,-80.295,169.225,36.966,156.954
C02487=1040.325,-21.053,-80.308,169.227,36.967,156.954
C02488=1040.331,-20.823,-80.321,169.229,36.967,156.954
C02489=1040.337,-20.594,-80.334,169.231,36.967,156.954
C02490=1040.342,-20.364,-80.347,169.233,36.968,156.954
C02491=1040.348,-20.134,-80.360,169.236,36.969,156.954
C02492=1040.354,-19.904,-80.373,169.238,36.969,156.954
C02493=1040.361,-19.674,-80.385,169.240,36.969,156.954
C02494=1040.367,-19.445,-80.398,169.242,36.970,156.954
C02495=1040.375,-19.071,-80.419,169.245,36.971,156.955
C02496=1040.386,-18.679,-80.441,169.248,36.972,156.955
C02497=1040.392,-18.429,-80.455,169.251,36.972,156.955
C02498=1040.398,-18.179,-80.469,169.253,36.973,156.955
C02499=1040.404,-17.930,-80.484,169.255,36.973,156.955
C02500=1040.411,-17.680,-80.497,169.257,36.974,156.955
C02501=1040.418,-17.431,-80.511,169.259,36.975,156.955
C02502=1040.424,-17.181,-80.525,169.261,36.975,156.955
C02503=1040.430,-16.932,-80.539,169.263,36.975,156.956
C02504=1040.436,-16.682,-80.554,169.266,36.976,156.956
C02505=1040.443,-16.433,-80.567,169.268,36.977,156.956
C02506=1040.450,-16.183,-80.581,169.270,36.977,156.956
C02507=1040.455,-15.934,-80.595,169.273,36.978,156.956
C02508=1040.462,-15.684,-80.609,169.275,36.978,156.956
C02509=1040.468,-15.434,-80.624,169.277,36.979,156.956
C02510=1040.475,-15.185,-80.638,169.279,36.980,156.956
C02511=1040.481,-14.935,-80.652,169.281,36.980,156.957
C02512=1040.487,-14.686,-80.667,169.283,36.981,156.957
C02513=1040.494,-14.436,-80.680,169.285,36.981,156.957
C02514=1040.499,-14.187,-80.695,169.287,36.982,156.957
C02515=1040.506,-13.937,-80.708,169.289,36.983,156.957
C02516=1040.513,-13.688,-80.723,169.292,36.983,156.957
C02517=1040.518,-13.438,-80.737,169.294,36.984,156.957
C02518=1040.525,-13.189,-80.752,169.296,36.985,156.957
C02519=1040.531,-12.940,-80.766,169.298,36.985,156.958
C02520=1040.537,-12.690,-80.780,169.300,36.986,156.958
C02521=1040.544,-12.440,-80.795,169.302,36.986,156.958
C02522=1040.550,-12.191,-80.809,169.304,36.987,156.958
C02523=1040.556,-11.941,-80.823,169.306,36.988,156.958
C02524=1040.563,-11.692,-80.837,169.308,36.988,156.958
C02525=1040.569,-11.442,-80.852,169.310,36.989,156.958
C02526=1040.575,-11.192,-80.867,169.312,36.990,156.959
C02527=1040.581,-10.944,-80.881,169.316,36.991,156.959
C02528=1040.588,-10.693,-80.895,169.318,36.991,156.959
C02529=1040.594,-10.444,-80.910,169.320,36.992,156.959
C02530=1040.600,-10.195,-80.924,169.322,36.993,156.959
C02531=1040.607,-9.945,-80.938,169.324,36.993,156.959
C02532=1040.613,-9.695,-80.953,169.326,36.994,156.959
C02533=1040.619,-9.447,-80.967,169.328,36.994,156.959
C02534=1040.626,-9.196,-80.981,169.330,36.995,156.960
C02535=1040.632,-8.947,-80.996,169.332,36.996,156.960
C02536=1040.638,-8.698,-81.011,169.334,36.996,156.960
C02537=1040.645,-8.448,-81.025,169.336,36.997,156.960
C02538=1040.651,-8.198,-81.039,169.338,36.997,156.960
C02539=1040.657,-7.949,-81.054,169.340,36.998,156.960
C02540=1040.664,-7.700,-81.068,169.343,36.999,156.960
C02541=1040.670,-7.450,-81.083,169.345,36.999,156.960
C02542=1040.676,-7.201,-81.097,169.347,37.000,156.961
C02543=1040.683,-6.951,-81.111,169.349,37.001,156.961
C02544=1040.689,-6.702,-81.126,169.351,37.001,156.961
C02545=1040.696,-6.452,-81.141,169.353,37.002,156.961
C02546=1040.701,-6.203,-81.156,169.355,37.002,156.961
C02547=1040.708,-5.953,-81.170,169.357,37.004,156.961
C02548=1040.715,-5.703,-81.184,169.359,37.004,156.961
C02549=1040.721,-5.454,-81.199,169.361,37.005,156.961
C02550=1040.727,-5.205,-81.213,169.363,37.006,156.962
C02551=1040.734,-4.955,-81.228,169.366,37.006,156.962
C02552=1040.740,-4.706,-81.243,169.368,37.007,156.962
C02553=1040.746,-4.455,-81.258,169.370,37.007,156.962
C02554=1040.753,-4.207,-81.271,169.372,37.008,156.962
C02555=1040.759,-3.957,-81.286,169.374,37.009,156.962
C02556=1040.766,-3.674,-81.303,169.377,37.009,156.962
C02557=1040.774,-3.391,-81.320,169.379,37.010,156.962
C02558=1040.781,-3.107,-81.337,169.381,37.011,156.963
C02559=1040.788,-2.823,-81.354,169.383,37.012,156.963
C02560=1040.793,-2.574,-81.368,169.385,37.012,156.963
C02561=1040.800,-2.324,-81.383,169.388,37.014,156.963
C02562=1040.806,-2.075,-81.398,169.390,37.014,156.963
C02563=1040.813,-1.825,-81.413,169.392,37.015,156.963
C02564=1040.818,-1.576,-81.428,169.394,37.015,156.964
C02565=1040.825,-1.326,-81.442,169.396,37.017,156.964
C02566=1040.831,-1.077,-81.457,169.398,37.017,156.964
C02567=1040.838,-0.828,-81.473,169.400,37.018,156.964
C02568=1040.844,-0.579,-81.488,169.402,37.018,156.964
C02569=1040.850,-0.329,-81.503,169.404,37.020,156.964
C02570=1040.856,-0.079,-81.518,169.406,37.020,156.965
C02571=1040.863,0.170,-81.532,169.409,37.021,156.965
C02572=1040.869,0.420,-81.547,169.411,37.022,156.965
C02573=1040.875,0.669,-81.562,169.413,37.023,156.965
C02574=1040.881,0.919,-81.577,169.415,37.023,156.965
C02575=1040.888,1.168,-81.592,169.417,37.024,156.965
C02576=1040.894,1.418,-81.607,169.419,37.025,156.965
C02577=1040.900,1.668,-81.622,169.421,37.025,156.966
C02578=1040.905,1.917,-81.637,169.422,37.027,156.966
C02579=1040.912,2.166,-81.653,169.424,37.027,156.966
C02580=1040.919,2.416,-81.668,169.426,37.028,156.966
C02581=1040.925,2.665,-81.683,169.429,37.028,156.966
C02582=1040.931,2.915,-81.697,169.431,37.030,156.966
C02583=1040.938,3.165,-81.712,169.433,37.030,156.967
C02584=1040.944,3.413,-81.727,169.435,37.031,156.967
C02585=1040.950,3.663,-81.742,169.437,37.031,156.967
C02586=1040.957,3.912,-81.758,169.439,37.033,156.967
C02587=1040.963,4.162,-81.773,169.441,37.033,156.967
C02588=1040.969,4.411,-81.788,169.443,37.034,156.967
C02589=1040.976,4.661,-81.802,169.445,37.035,156.967
C02590=1040.982,4.911,-81.817,169.447,37.035,156.967
C02591=1040.989,5.160,-81.833,169.450,37.036,156.968
C02592=1040.994,5.409,-81.848,169.452,37.037,156.968
C02593=1041.000,5.659,-81.863,169.454,37.038,156.968
C02594=1041.007,5.908,-81.878,169.456,37.038,156.968
C02595=1041.013,6.157,-81.894,169.458,37.040,156.968
C02596=1041.020,6.407,-81.909,169.459,37.040,156.968
C02597=1041.026,6.657,-81.924,169.461,37.041,156.969
C02598=1041.032,6.906,-81.939,169.463,37.041,156.969
C02599=1041.039,7.155,-81.954,169.465,37.042,156.969
C02600=1041.046,7.405,-81.969,169.467,37.043,156.969
C02601=1041.052,7.655,-81.984,169.470,37.044,156.969
C02602=1041.059,7.904,-82.000,169.472,37.044,156.969
C02603=1041.064,8.154,-82.015,169.474,37.045,156.969
C02604=1041.070,8.403,-82.030,169.476,37.046,156.970
C02605=1041.077,8.652,-82.046,169.478,37.047,156.970
C02606=1041.083,8.901,-82.061,169.480,37.048,156.970
C02607=1041.089,9.151,-82.076,169.482,37.048,156.970
C02608=1041.096,9.400,-82.091,169.484,37.049,156.970
C02609=1041.103,9.650,-82.106,169.486,37.050,156.970
C02610=1041.109,9.899,-82.121,169.488,37.051,156.971
C02611=1041.116,10.148,-82.137,169.491,37.051,156.971
C02612=1041.121,10.398,-82.152,169.492,37.052,156.971
C02613=1041.128,10.648,-82.167,169.494,37.052,156.971
C02614=1041.134,10.897,-82.183,169.496,37.054,156.971
C02615=1041.141,11.147,-82.198,169.498,37.054,156.971
C02616=1041.147,11.396,-82.213,169.500,37.055,156.971
C02617=1041.154,11.645,-82.228,169.502,37.056,156.972
C02618=1041.160,11.895,-82.243,169.504,37.056,156.972
C02619=1041.167,12.144,-82.259,169.506,37.057,156.972
C02620=1041.174,12.429,-82.277,169.508,37.058,156.972
C02621=1041.181,12.716,-82.294,169.511,37.059,156.972
C02622=1041.188,13.001,-82.312,169.514,37.060,156.972
C02623=1041.196,13.286,-82.330,169.516,37.060,156.973
C02624=1041.202,13.536,-82.345,169.518,37.061,156.973
C02625=1041.209,13.785,-82.360,169.520,37.062,156.973
C02626=1041.215,14.034,-82.375,169.522,37.063,156.973
C02627=1041.221,14.284,-82.391,169.523,37.064,156.973
C02628=1041.228,14.533,-82.407,169.525,37.064,156.973
C02629=1041.234,14.782,-82.422,169.527,37.065,156.974
C02630=1041.240,15.032,-82.438,169.530,37.066,156.974
C02631=1041.247,15.281,-82.453,169.532,37.067,156.974
C02632=1041.253,15.530,-82.469,169.534,37.068,156.974
C02633=1041.260,15.781,-82.485,169.536,37.068,156.974
C02634=1041.266,16.030,-82.500,169.538,37.069,156.974
C02635=1041.272,16.279,-82.517,169.539,37.070,156.974
C02636=1041.279,16.529,-82.532,169.541,37.071,156.975
C02637=1041.285,16.778,-82.547,169.543,37.072,156.975
C02638=1041.291,17.028,-82.563,169.545,37.073,156.975
C02639=1041.298,17.277,-82.579,169.548,37.073,156.975
C02640=1041.304,17.526,-82.595,169.550,37.074,156.975
C02641=1041.310,17.776,-82.610,169.552,37.075,156.975
C02642=1041.317,18.025,-82.625,169.554,37.076,156.976
C02643=1041.323,18.275,-82.642,169.556,37.076,156.976
C02644=1041.329,18.524,-82.657,169.557,37.078,156.976
C02645=1041.335,18.774,-82.673,169.559,37.078,156.976
C02646=1041.342,19.023,-82.689,169.561,37.079,156.976
C02647=1041.349,19.273,-82.704,169.563,37.080,156.976
C02648=1041.355,19.522,-82.720,169.566,37.081,156.977
C02649=1041.361,19.771,-82.736,169.568,37.081,156.977
C02650=1041.367,20.021,-82.752,169.570,37.083,156.977
C02651=1041.374,20.270,-82.767,169.572,37.083,156.977
C02652=1041.380,20.520,-82.783,169.573,37.085,156.977
C02653=1041.386,20.769,-82.799,169.575,37.085,156.977
C02654=1041.392,21.018,-82.815,169.577,37.086,156.978
C02655=1041.399,21.268,-82.830,169.579,37.087,156.978
C02656=1041.405,21.518,-82.847,169.581,37.088,156.978
C02657=1041.412,21.767,-82.862,169.584,37.089,156.978
C02658=1041.418,22.016,-82.879,169.586,37.089,156.978
C02659=1041.425,22.265,-82.894,169.587,37.090,156.978
C02660=1041.430,22.515,-82.910,169.589,37.091,156.979
C02661=1041.437,22.764,-82.925,169.591,37.092,156.979
C02662=1041.443,23.014,-82.942,169.593,37.093,156.979
C02663=1041.449,23.263,-82.958,169.595,37.094,156.979
C02664=1041.456,23.513,-82.974,169.597,37.094,156.979
C02665=1041.462,23.762,-82.990,169.600,37.096,156.980
C02666=1041.468,24.012,-83.005,169.601,37.096,156.980
C02667=1041.474,24.261,-83.021,169.603,37.098,156.980
C02668=1041.481,24.510,-83.037,169.605,37.098,156.980
C02669=1041.487,24.759,-83.053,169.607,37.099,156.980
C02670=1041.494,25.009,-83.069,169.609,37.100,156.980
C02671=1041.500,25.258,-83.086,169.611,37.101,156.981
C02672=1041.506,25.508,-83.102,169.612,37.101,156.981
C02673=1041.513,25.757,-83.118,169.615,37.102,156.981
C02674=1041.519,26.006,-83.134,169.617,37.103,156.981
C02675=1041.526,26.256,-83.150,169.619,37.104,156.981
C02676=1041.532,26.505,-83.166,169.621,37.105,156.981
C02677=1041.538,26.755,-83.182,169.623,37.105,156.982
C02678=1041.544,27.004,-83.197,169.625,37.107,156.982
C02679=1041.550,27.254,-83.214,169.626,37.107,156.982
C02680=1041.558,27.503,-83.230,169.628,37.109,156.982
C02681=1041.564,27.753,-83.246,169.630,37.109,156.982
C02682=1041.570,28.002,-83.262,169.633,37.110,156.982
C02683=1041.576,28.251,-83.278,169.635,37.111,156.983
C02684=1041.584,28.538,-83.297,169.637,37.112,156.983
C02685=1041.591,28.825,-83.316,169.639,37.113,156.983
C02686=1041.598,29.111,-83.334,169.641,37.114,156.983
C02687=1041.605,29.398,-83.353,169.643,37.115,156.983
C02688=1041.611,29.647,-83.369,169.645,37.116,156.984
C02689=1041.618,29.897,-83.386,169.648,37.117,156.984
C02690=1041.624,30.146,-83.402,169.650,37.118,156.984
C02691=1041.630,30.396,-83.418,169.651,37.119,156.984
C02692=1041.637,30.644,-83.434,169.653,37.120,156.984
C02693=1041.643,30.894,-83.451,169.655,37.121,156.985
C02694=1041.649,31.144,-83.467,169.657,37.122,156.985
C02695=1041.655,31.393,-83.484,169.659,37.122,156.985
C02696=1041.661,31.642,-83.500,169.660,37.123,156.985
C02697=1041.668,31.892,-83.516,169.662,37.124,156.985
C02698=1041.674,32.141,-83.532,169.665,37.125,156.985
C02699=1041.681,32.390,-83.549,169.667,37.126,156.986
C02700=1041.687,32.640,-83.565,169.669,37.127,156.986
C02701=1041.693,32.890,-83.582,169.671,37.128,156.986
C02702=1041.700,33.139,-83.598,169.672,37.129,156.986
C02703=1041.706,33.388,-83.614,169.674,37.130,156.986
C02704=1041.712,33.638,-83.630,169.676,37.131,156.987
C02705=1041.719,33.887,-83.647,169.678,37.131,156.987
C02706=1041.725,34.136,-83.664,169.681,37.133,156.987
C02707=1041.731,34.385,-83.679,169.682,37.133,156.987
C02708=1041.738,34.635,-83.696,169.684,37.134,156.987
C02709=1041.744,34.885,-83.712,169.686,37.135,156.987
C02710=1041.750,35.133,-83.729,169.688,37.136,156.988
C02711=1041.757,35.383,-83.746,169.690,37.137,156.988
C02712=1041.763,35.632,-83.761,169.691,37.138,156.988
C02713=1041.769,35.882,-83.778,169.693,37.139,156.988
C02714=1041.776,36.131,-83.795,169.696,37.139,156.988
C02715=1041.782,36.380,-83.811,169.698,37.141,156.989
C02716=1041.789,36.631,-83.828,169.700,37.141,156.989
C02717=1041.795,36.879,-83.845,169.702,37.142,156.989
C02718=1041.802,37.128,-83.861,169.703,37.143,156.989
C02719=1041.808,37.378,-83.877,169.705,37.144,156.989
C02720=1041.814,37.628,-83.893,169.707,37.145,156.989
C02721=1041.820,37.876,-83.910,169.710,37.146,156.990
C02722=1041.827,38.126,-83.927,169.712,37.147,156.990
C02723=1041.833,38.375,-83.944,169.713,37.148,156.990
C02724=1041.839,38.625,-83.960,169.715,37.149,156.990
C02725=1041.846,38.875,-83.977,169.717,37.150,156.990
C02726=1041.851,39.124,-83.994,169.719,37.150,156.991
C02727=1041.857,39.373,-84.011,169.720,37.152,156.991
C02728=1041.864,39.622,-84.028,169.722,37.153,156.991
C02729=1041.870,39.872,-84.044,169.725,37.154,156.991
C02730=1041.876,40.122,-84.061,169.727,37.155,156.991
C02731=1041.883,40.371,-84.078,169.729,37.155,156.991
C02732=1041.889,40.620,-84.094,169.730,37.157,156.992
C02733=1041.896,40.869,-84.112,169.732,37.157,156.992
C02734=1041.901,41.119,-84.128,169.734,37.158,156.992
C02735=1041.908,41.367,-84.145,169.736,37.159,156.992
C02736=1041.914,41.617,-84.161,169.737,37.160,156.992
C02737=1041.921,41.866,-84.178,169.740,37.162,156.993
C02738=1041.927,42.116,-84.195,169.742,37.162,156.993
C02739=1041.933,42.365,-84.212,169.744,37.163,156.993
C02740=1041.940,42.615,-84.229,169.746,37.164,156.993
C02741=1041.946,42.864,-84.246,169.747,37.165,156.993
C02742=1041.952,43.113,-84.262,169.749,37.166,156.994
C02743=1041.959,43.362,-84.279,169.751,37.167,156.994
C02744=1041.964,43.612,-84.296,169.754,37.168,156.994
C02745=1041.971,43.862,-84.313,169.755,37.169,156.994
C02746=1041.977,44.111,-84.330,169.757,37.170,156.994
C02747=1041.983,44.360,-84.347,169.759,37.171,156.995
C02748=1041.990,44.647,-84.367,169.761,37.173,156.995
C02749=1041.997,44.933,-84.386,169.763,37.173,156.995
C02750=1042.004,45.219,-84.405,169.765,37.174,156.995
C02751=1042.011,45.507,-84.425,169.768,37.176,156.996
C02752=1042.017,45.756,-84.443,169.770,37.177,156.996
C02753=1042.024,46.005,-84.460,169.771,37.178,156.996
C02754=1042.030,46.255,-84.476,169.773,37.179,156.996
C02755=1042.036,46.504,-84.494,169.775,37.180,156.996
C02756=1042.042,46.753,-84.511,169.777,37.181,156.997
C02757=1042.048,47.002,-84.527,169.778,37.182,156.997
C02758=1042.055,47.252,-84.545,169.781,37.183,156.997
C02759=1042.060,47.501,-84.562,169.783,37.184,156.997
C02760=1042.067,47.751,-84.579,169.785,37.185,156.997
C02761=1042.073,48.000,-84.596,169.786,37.186,156.998
C02762=1042.079,48.249,-84.614,169.788,37.187,156.998
C02763=1042.086,48.498,-84.631,169.790,37.188,156.998
C02764=1042.092,48.748,-84.647,169.792,37.189,156.998
C02765=1042.098,48.997,-84.665,169.794,37.190,156.999
C02766=1042.105,49.247,-84.682,169.796,37.191,156.999
C02767=1042.111,49.495,-84.699,169.798,37.192,156.999
C02768=1042.117,49.746,-84.716,169.800,37.193,156.999
C02769=1042.123,49.994,-84.733,169.801,37.194,156.999
C02770=1042.130,50.244,-84.751,169.803,37.195,157.000
C02771=1042.135,50.493,-84.768,169.805,37.196,157.000
C02772=1042.142,50.743,-84.785,169.808,37.197,157.000
C02773=1042.147,50.992,-84.802,169.809,37.198,157.000
C02774=1042.154,51.241,-84.820,169.811,37.199,157.000
C02775=1042.160,51.490,-84.837,169.813,37.200,157.001
C02776=1042.167,51.740,-84.855,169.815,37.202,157.001
C02777=1042.173,51.989,-84.872,169.816,37.202,157.001
C02778=1042.179,52.239,-84.888,169.818,37.203,157.001
C02779=1042.185,52.488,-84.906,169.821,37.204,157.001
C02780=1042.192,52.737,-84.923,169.823,37.205,157.002
C02781=1042.198,52.986,-84.940,169.824,37.206,157.002
C02782=1042.204,53.236,-84.958,169.826,37.207,157.002
C02783=1042.211,53.485,-84.975,169.828,37.208,157.002
C02784=1042.217,53.734,-84.992,169.830,37.210,157.002
C02785=1042.223,53.984,-85.010,169.832,37.210,157.003
C02786=1042.229,54.233,-85.027,169.834,37.211,157.003
C02787=1042.235,54.483,-85.045,169.836,37.212,157.003
C02788=1042.242,54.732,-85.062,169.838,37.213,157.003
C02789=1042.249,54.981,-85.079,169.840,37.214,157.003
C02790=1042.255,55.230,-85.097,169.841,37.215,157.003
C02791=1042.261,55.479,-85.114,169.843,37.216,157.004
C02792=1042.268,55.729,-85.131,169.845,37.217,157.004
C02793=1042.274,55.978,-85.149,169.848,37.218,157.004
C02794=1042.280,56.227,-85.166,169.849,37.219,157.004
C02795=1042.286,56.477,-85.184,169.851,37.220,157.004
C02796=1042.293,56.726,-85.201,169.853,37.221,157.005
C02797=1042.299,56.975,-85.218,169.855,37.222,157.005
C02798=1042.305,57.225,-85.236,169.856,37.223,157.005
C02799=1042.312,57.473,-85.253,169.858,37.224,157.005
C02800=1042.318,57.723,-85.271,169.861,37.225,157.005
C02801=1042.325,57.973,-85.288,169.863,37.226,157.006
C02802=1042.331,58.221,-85.305,169.864,37.227,157.006
C02803=1042.337,58.471,-85.323,169.866,37.228,157.006
C02804=1042.344,58.721,-85.341,169.868,37.229,157.006
C02805=1042.349,58.970,-85.358,169.870,37.230,157.006
C02806=1042.356,59.219,-85.376,169.871,37.231,157.007
C02807=1042.363,59.468,-85.393,169.873,37.232,157.007
C02808=1042.369,59.717,-85.410,169.876,37.233,157.007
C02809=1042.376,59.967,-85.428,169.878,37.233,157.007
C02810=1042.382,60.217,-85.446,169.879,37.235,157.007
C02811=1042.388,60.465,-85.463,169.881,37.236,157.008
C02812=1042.396,60.752,-85.483,169.883,37.236,157.008
C02813=1042.402,61.038,-85.503,169.885,37.238,157.008
C02814=1042.410,61.325,-85.523,169.888,37.239,157.008
C02815=1042.418,61.611,-85.544,169.890,37.240,157.009
C02816=1042.424,61.860,-85.561,169.892,37.241,157.009
C02817=1042.430,62.110,-85.579,169.894,37.242,157.009
C02818=1042.437,62.358,-85.597,169.896,37.243,157.009
C02819=1042.443,62.607,-85.614,169.897,37.244,157.009
C02820=1042.450,62.857,-85.631,169.899,37.245,157.010
C02821=1042.456,63.106,-85.649,169.901,37.246,157.010
C02822=1042.463,63.356,-85.667,169.904,37.247,157.010
C02823=1042.469,63.605,-85.684,169.905,37.247,157.010
C02824=1042.475,63.855,-85.702,169.907,37.249,157.010
C02825=1042.482,64.103,-85.720,169.909,37.249,157.010
C02826=1042.488,64.353,-85.738,169.911,37.250,157.011
C02827=1042.494,64.602,-85.755,169.912,37.252,157.011
C02828=1042.501,64.852,-85.773,169.915,37.253,157.011
C02829=1042.507,65.101,-85.791,169.917,37.254,157.011
C02830=1042.513,65.350,-85.809,169.919,37.255,157.012
C02831=1042.519,65.599,-85.826,169.920,37.256,157.012
C02832=1042.525,65.849,-85.844,169.922,37.257,157.012
C02833=1042.532,66.098,-85.863,169.924,37.258,157.012
C02834=1042.539,66.348,-85.880,169.925,37.259,157.012
C02835=1042.544,66.597,-85.898,169.928,37.260,157.013
C02836=1042.551,66.846,-85.916,169.930,37.261,157.013
C02837=1042.557,67.095,-85.934,169.932,37.262,157.013
C02838=1042.564,67.345,-85.952,169.933,37.263,157.013
C02839=1042.570,67.593,-85.970,169.935,37.264,157.013
C02840=1042.576,67.843,-85.988,169.937,37.265,157.014
C02841=1042.582,68.093,-86.006,169.939,37.266,157.014
C02842=1042.589,68.342,-86.024,169.941,37.267,157.014
C02843=1042.594,68.591,-86.041,169.943,37.268,157.014
C02844=1042.601,68.840,-86.060,169.945,37.269,157.015
C02845=1042.607,69.089,-86.078,169.947,37.270,157.015
C02846=1042.614,69.339,-86.095,169.948,37.271,157.015
C02847=1042.620,69.588,-86.114,169.950,37.272,157.015
C02848=1042.626,69.837,-86.131,169.953,37.274,157.015
C02849=1042.632,70.086,-86.150,169.954,37.274,157.016
C02850=1042.638,70.336,-86.168,169.956,37.276,157.016
C02851=1042.645,70.585,-86.187,169.958,37.277,157.016
C02852=1042.651,70.834,-86.204,169.960,37.278,157.016
C02853=1042.657,71.084,-86.222,169.961,37.279,157.016
C02854=1042.664,71.333,-86.240,169.963,37.280,157.017
C02855=1042.670,71.582,-86.258,169.966,37.281,157.017
C02856=1042.676,71.831,-86.277,169.968,37.282,157.017
C02857=1042.682,72.081,-86.294,169.969,37.283,157.017
C02858=1042.688,72.330,-86.313,169.971,37.284,157.018
C02859=1042.694,72.579,-86.331,169.973,37.285,157.018
C02860=1042.701,72.829,-86.350,169.974,37.287,157.018
C02861=1042.707,73.078,-86.368,169.976,37.287,157.018
C02862=1042.714,73.327,-86.386,169.979,37.288,157.018
C02863=1042.720,73.575,-86.404,169.981,37.290,157.019
C02864=1042.726,73.825,-86.422,169.982,37.291,157.019
C02865=1042.732,74.074,-86.440,169.984,37.291,157.019
C02866=1042.738,74.324,-86.458,169.986,37.293,157.019
C02867=1042.745,74.573,-86.477,169.987,37.294,157.020
C02868=1042.751,74.822,-86.496,169.990,37.295,157.020
C02869=1042.757,75.072,-86.514,169.992,37.296,157.020
C02870=1042.763,75.320,-86.532,169.994,37.297,157.020
C02871=1042.769,75.570,-86.550,169.995,37.298,157.020
C02872=1042.776,75.819,-86.568,169.997,37.299,157.021
C02873=1042.782,76.068,-86.587,169.999,37.300,157.021
C02874=1042.788,76.318,-86.605,170.002,37.301,157.021
C02875=1042.795,76.567,-86.624,170.003,37.302,157.021
C02876=1042.802,76.853,-86.644,170.005,37.304,157.022
C02877=1042.809,77.140,-86.665,170.007,37.305,157.022
C02878=1042.817,77.426,-86.686,170.009,37.306,157.022
C02879=1042.823,77.711,-86.708,170.011,37.307,157.022
C02880=1042.830,77.960,-86.726,170.013,37.308,157.022
C02881=1042.836,78.210,-86.744,170.016,37.309,157.023
C02882=1042.842,78.459,-86.763,170.017,37.310,157.023
C02883=1042.849,78.708,-86.781,170.019,37.312,157.023
C02884=1042.855,78.957,-86.800,170.021,37.313,157.023
C02885=1042.861,79.207,-86.818,170.023,37.314,157.024
C02886=1042.867,79.457,-86.837,170.024,37.315,157.024
C02887=1042.873,79.705,-86.856,170.027,37.316,157.024
C02888=1042.879,79.954,-86.874,170.029,37.317,157.024
C02889=1042.885,80.203,-86.893,170.030,37.318,157.025
C02890=1042.892,80.453,-86.911,170.032,37.319,157.025
C02891=1042.897,80.702,-86.930,170.034,37.321,157.025
C02892=1042.904,80.952,-86.949,170.035,37.321,157.025
C02893=1042.910,81.201,-86.967,170.038,37.323,157.025
C02894=1042.917,81.450,-86.986,170.040,37.324,157.026
C02895=1042.923,81.699,-87.005,170.042,37.325,157.026
C02896=1042.928,81.949,-87.023,170.043,37.326,157.026
C02897=1042.935,82.198,-87.042,170.045,37.327,157.026
C02898=1042.941,82.447,-87.060,170.047,37.328,157.027
C02899=1042.947,82.696,-87.079,170.049,37.329,157.027
C02900=1042.953,82.945,-87.097,170.051,37.330,157.027
C02901=1042.959,83.194,-87.117,170.053,37.332,157.027
C02902=1042.966,83.443,-87.135,170.055,37.333,157.028
C02903=1042.972,83.692,-87.154,170.056,37.334,157.028
C02904=1042.978,83.942,-87.173,170.058,37.335,157.028
C02905=1042.985,84.191,-87.191,170.061,37.336,157.028
C02906=1042.990,84.441,-87.210,170.063,37.337,157.028
C02907=1042.997,84.690,-87.228,170.064,37.338,157.029
C02908=1043.003,84.939,-87.247,170.066,37.340,157.029
C02909=1043.010,85.188,-87.266,170.068,37.340,157.029
C02910=1043.015,85.438,-87.285,170.069,37.341,157.029
C02911=1043.022,85.687,-87.304,170.072,37.343,157.030
C02912=1043.028,85.936,-87.322,170.074,37.344,157.030
C02913=1043.035,86.185,-87.341,170.076,37.345,157.030
C02914=1043.041,86.434,-87.360,170.077,37.346,157.030
C02915=1043.047,86.684,-87.379,170.079,37.347,157.030
C02916=1043.053,86.933,-87.397,170.081,37.348,157.031
C02917=1043.059,87.182,-87.416,170.084,37.349,157.031
C02918=1043.066,87.431,-87.435,170.085,37.350,157.031
C02919=1043.072,87.680,-87.454,170.087,37.351,157.031
C02920=1043.078,87.929,-87.473,170.089,37.352,157.032
C02921=1043.084,88.179,-87.491,170.091,37.354,157.032
C02922=1043.091,88.428,-87.510,170.092,37.355,157.032
C02923=1043.097,88.677,-87.529,170.094,37.355,157.032
C02924=1043.104,88.927,-87.548,170.097,37.357,157.032
C02925=1043.110,89.176,-87.567,170.098,37.358,157.033
C02926=1043.116,89.425,-87.585,170.100,37.359,157.033
C02927=1043.122,89.675,-87.605,170.102,37.360,157.033
C02928=1043.129,89.923,-87.624,170.104,37.361,157.033
C02929=1043.135,90.172,-87.643,170.105,37.362,157.034
C02930=1043.141,90.422,-87.662,170.108,37.363,157.034
C02931=1043.147,90.671,-87.681,170.110,37.364,157.034
C02932=1043.153,90.920,-87.700,170.112,37.366,157.034
C02933=1043.160,91.169,-87.719,170.113,37.367,157.035
C02934=1043.165,91.419,-87.738,170.115,37.368,157.035
C02935=1043.172,91.667,-87.757,170.117,37.369,157.035
C02936=1043.178,91.917,-87.776,170.119,37.370,157.035
C02937=1043.184,92.166,-87.795,170.121,37.371,157.036
C02938=1043.190,92.415,-87.814,170.123,37.372,157.036
C02939=1043.196,92.664,-87.834,170.125,37.374,157.036
C02940=1043.204,92.950,-87.855,170.127,37.375,157.036
C02941=1043.211,93.236,-87.877,170.130,37.376,157.037
C02942=1043.217,93.522,-87.900,170.132,37.378,157.037
C02943=1043.225,93.809,-87.921,170.134,37.379,157.037
C02944=1043.231,94.057,-87.941,170.135,37.380,157.037
C02945=1043.237,94.307,-87.960,170.137,37.382,157.038
C02946=1043.243,94.556,-87.979,170.139,37.382,157.038
C02947=1043.249,94.805,-87.998,170.141,37.383,157.038
C02948=1043.256,95.054,-88.017,170.143,37.385,157.038
C02949=1043.262,95.304,-88.037,170.145,37.386,157.039
C02950=1043.268,95.553,-88.056,170.147,37.387,157.039
C02951=1043.275,95.802,-88.076,170.148,37.388,157.039
C02952=1043.280,96.051,-88.095,170.151,37.389,157.039
C02953=1043.287,96.300,-88.113,170.153,37.391,157.040
C02954=1043.293,96.549,-88.133,170.155,37.391,157.040
C02955=1043.299,96.798,-88.152,170.156,37.392,157.040
C02956=1043.305,97.048,-88.172,170.158,37.394,157.040
C02957=1043.312,97.297,-88.191,170.160,37.395,157.040
C02958=1043.318,97.546,-88.210,170.163,37.396,157.041
C02959=1043.324,97.795,-88.229,170.164,37.397,157.041
C02960=1043.330,98.044,-88.249,170.166,37.399,157.041
C02961=1043.337,98.293,-88.267,170.168,37.400,157.041
C02962=1043.343,98.543,-88.288,170.170,37.400,157.042
C02963=1043.349,98.792,-88.307,170.171,37.402,157.042
C02964=1043.355,99.041,-88.326,170.174,37.403,157.042
C02965=1043.361,99.290,-88.346,170.176,37.404,157.042
C02966=1043.368,99.539,-88.364,170.177,37.405,157.043
C02967=1043.374,99.789,-88.385,170.179,37.406,157.043
C02968=1043.381,100.038,-88.403,170.181,37.407,157.043
C02969=1043.387,100.287,-88.423,170.183,37.408,157.043
C02970=1043.392,100.536,-88.443,170.186,37.409,157.043
C02971=1043.399,100.785,-88.462,170.187,37.411,157.044
C02972=1043.405,101.035,-88.481,170.189,37.412,157.044
C02973=1043.411,101.284,-88.501,170.191,37.413,157.044
C02974=1043.417,101.533,-88.521,170.192,37.414,157.044
C02975=1043.423,101.782,-88.541,170.194,37.415,157.045
C02976=1043.430,102.031,-88.559,170.197,37.417,157.045
C02977=1043.436,102.280,-88.579,170.199,37.418,157.045
C02978=1043.442,102.529,-88.600,170.200,37.419,157.045
C02979=1043.448,102.779,-88.619,170.202,37.420,157.046
C02980=1043.454,103.028,-88.639,170.204,37.422,157.046
C02981=1043.460,103.277,-88.658,170.207,37.423,157.046
C02982=1043.466,103.526,-88.677,170.208,37.424,157.046
C02983=1043.473,103.775,-88.698,170.210,37.425,157.047
C02984=1043.479,104.025,-88.717,170.212,37.426,157.047
C02985=1043.485,104.273,-88.737,170.213,37.428,157.047
C02986=1043.490,104.523,-88.756,170.216,37.429,157.047
C02987=1043.498,104.772,-88.776,170.218,37.430,157.048
C02988=1043.504,105.021,-88.796,170.220,37.431,157.048
C02989=1043.509,105.270,-88.815,170.221,37.432,157.048
C02990=1043.515,105.519,-88.835,170.223,37.434,157.048
C02991=1043.522,105.769,-88.855,170.225,37.435,157.049
C02992=1043.528,106.018,-88.875,170.228,37.435,157.049
C02993=1043.534,106.267,-88.894,170.229,37.437,157.049
C02994=1043.540,106.515,-88.914,170.231,37.438,157.049
C02995=1043.547,106.765,-88.934,170.233,37.439,157.050
C02996=1043.553,107.014,-88.954,170.235,37.440,157.050
C02997=1043.559,107.263,-88.973,170.237,37.441,157.050
C02998=1043.565,107.512,-88.993,170.239,37.443,157.050
C02999=1043.572,107.762,-89.012,170.241,37.444,157.051
C03000=1043.578,108.011,-89.032,170.243,37.445,157.051
C03001=1043.584,108.259,-89.052,170.245,37.446,157.051
C03002=1043.590,108.509,-89.073,170.246,37.448,157.051
C03003=1043.596,108.758,-89.092,170.249,37.449,157.052
C03004=1043.603,109.044,-89.114,170.251,37.450,157.052
C03005=1043.610,109.330,-89.137,170.253,37.451,157.052
C03006=1043.617,109.617,-89.161,170.255,37.452,157.052
C03007=1043.625,109.902,-89.184,170.257,37.454,157.053
C03008=1043.631,110.151,-89.203,170.260,37.455,157.053
C03009=1043.637,110.400,-89.223,170.262,37.457,157.053
C03010=1043.643,110.650,-89.243,170.264,37.457,157.053
C03011=1043.649,110.898,-89.263,170.265,37.458,157.054
C03012=1043.655,111.147,-89.283,170.267,37.460,157.054
C03013=1043.662,111.397,-89.303,170.269,37.461,157.054
C03014=1043.668,111.646,-89.323,170.272,37.462,157.054
C03015=1043.674,111.895,-89.343,170.273,37.463,157.055
C03016=1043.680,112.145,-89.363,170.275,37.464,157.055
C03017=1043.686,112.393,-89.383,170.277,37.466,157.055
C03018=1043.693,112.643,-89.403,170.279,37.467,157.055
C03019=1043.699,112.892,-89.423,170.281,37.468,157.056
C03020=1043.705,113.140,-89.443,170.283,37.469,157.056
C03021=1043.711,113.390,-89.463,170.285,37.470,157.056
C03022=1043.717,113.639,-89.483,170.287,37.472,157.056
C03023=1043.723,113.888,-89.503,170.288,37.473,157.057
C03024=1043.730,114.137,-89.524,170.291,37.475,157.057
C03025=1043.735,114.386,-89.544,170.293,37.476,157.057
C03026=1043.741,114.635,-89.564,170.295,37.477,157.058
C03027=1043.748,114.885,-89.584,170.296,37.478,157.058
C03028=1043.754,115.133,-89.604,170.298,37.480,157.058
C03029=1043.759,115.383,-89.625,170.300,37.481,157.058
C03030=1043.766,115.632,-89.645,170.303,37.482,157.059
C03031=1043.772,115.881,-89.665,170.304,37.483,157.059
C03032=1043.777,116.130,-89.686,170.306,37.485,157.059
C03033=1043.783,116.379,-89.706,170.308,37.486,157.060
C03034=1043.789,116.628,-89.726,170.311,37.487,157.060
C03035=1043.796,116.876,-89.747,170.313,37.489,157.060
C03036=1043.802,117.126,-89.768,170.314,37.490,157.060
C03037=1043.808,117.375,-89.788,170.316,37.491,157.061
C03038=1043.814,117.625,-89.808,170.318,37.492,157.061
C03039=1043.819,117.874,-89.829,170.320,37.493,157.061
C03040=1043.825,118.123,-89.848,170.322,37.495,157.061
C03041=1043.832,118.372,-89.869,170.324,37.496,157.062
C03042=1043.838,118.621,-89.889,170.326,37.498,157.062
C03043=1043.844,118.870,-89.910,170.328,37.499,157.062
C03044=1043.850,119.119,-89.930,170.329,37.500,157.062
C03045=1043.856,119.368,-89.950,170.332,37.501,157.063
C03046=1043.862,119.618,-89.971,170.334,37.502,157.063
C03047=1043.868,119.866,-89.991,170.336,37.504,157.063
C03048=1043.875,120.115,-90.012,170.338,37.505,157.063
C03049=1043.880,120.364,-90.033,170.339,37.506,157.064
C03050=1043.887,120.614,-90.053,170.342,37.507,157.064
C03051=1043.893,120.863,-90.073,170.344,37.509,157.064
C03052=1043.899,121.112,-90.093,170.346,37.510,157.065
C03053=1043.905,121.361,-90.115,170.348,37.511,157.065
C03054=1043.911,121.610,-90.135,170.349,37.513,157.065
C03055=1043.917,121.859,-90.155,170.352,37.514,157.065
C03056=1043.923,122.108,-90.176,170.354,37.515,157.066
C03057=1043.930,122.357,-90.197,170.356,37.516,157.066
C03058=1043.936,122.606,-90.217,170.357,37.518,157.066
C03059=1043.942,122.856,-90.237,170.359,37.519,157.066
C03060=1043.948,123.104,-90.258,170.362,37.520,157.067
C03061=1043.954,123.353,-90.278,170.364,37.521,157.067
C03062=1043.960,123.603,-90.299,170.366,37.522,157.067
C03063=1043.967,123.851,-90.320,170.368,37.523,157.067
C03064=1043.973,124.100,-90.340,170.369,37.525,157.068
C03065=1043.978,124.350,-90.361,170.372,37.527,157.068
C03066=1043.985,124.598,-90.382,170.374,37.528,157.068
C03067=1043.991,124.848,-90.402,170.376,37.529,157.069
C03068=1043.998,125.133,-90.426,170.378,37.530,157.069
C03069=1044.006,125.420,-90.449,170.380,37.531,157.069
C03070=1044.012,125.706,-90.473,170.383,37.533,157.069
C03071=1044.019,125.992,-90.497,170.385,37.534,157.070
C03072=1044.025,126.241,-90.517,170.387,37.536,157.070
C03073=1044.032,126.489,-90.538,170.389,37.537,157.070
C03074=1044.038,126.739,-90.559,170.391,37.538,157.071
C03075=1044.045,126.987,-90.580,170.393,37.539,157.071
C03076=1044.051,127.236,-90.600,170.395,37.541,157.071
C03077=1044.056,127.486,-90.621,170.397,37.542,157.071
C03078=1044.063,127.735,-90.642,170.399,37.543,157.072
C03079=1044.069,127.984,-90.662,170.401,37.545,157.072
C03080=1044.075,128.233,-90.683,170.404,37.546,157.072
C03081=1044.081,128.482,-90.703,170.405,37.547,157.072
C03082=1044.088,128.731,-90.725,170.407,37.548,157.073
C03083=1044.094,128.981,-90.745,170.409,37.549,157.073
C03084=1044.101,129.229,-90.766,170.411,37.550,157.073
C03085=1044.106,129.479,-90.787,170.414,37.552,157.073
C03086=1044.113,129.727,-90.807,170.416,37.553,157.074
C03087=1044.119,129.976,-90.828,170.418,37.554,157.074
C03088=1044.125,130.225,-90.849,170.419,37.555,157.074
C03089=1044.131,130.474,-90.869,170.421,37.556,157.074
C03090=1044.138,130.723,-90.890,170.424,37.558,157.075
C03091=1044.144,130.973,-90.911,170.426,37.559,157.075
C03092=1044.150,131.221,-90.932,170.428,37.560,157.075
C03093=1044.157,131.470,-90.954,170.430,37.562,157.076
C03094=1044.162,131.720,-90.975,170.431,37.563,157.076
C03095=1044.169,131.968,-90.995,170.434,37.564,157.076
C03096=1044.175,132.218,-91.016,170.436,37.565,157.076
C03097=1044.181,132.467,-91.038,170.438,37.567,157.077
C03098=1044.187,132.716,-91.058,170.440,37.568,157.077
C03099=1044.193,132.965,-91.079,170.442,37.570,157.077
C03100=1044.199,133.214,-91.101,170.445,37.571,157.078
C03101=1044.205,133.463,-91.122,170.446,37.572,157.078
C03102=1044.212,133.712,-91.143,170.448,37.573,157.078
C03103=1044.217,133.961,-91.164,170.450,37.574,157.078
C03104=1044.224,134.210,-91.185,170.453,37.576,157.079
C03105=1044.230,134.459,-91.207,170.455,37.577,157.079
C03106=1044.235,134.708,-91.227,170.457,37.579,157.079
C03107=1044.242,134.957,-91.248,170.458,37.580,157.079
C03108=1044.248,135.207,-91.270,170.460,37.581,157.080
C03109=1044.254,135.455,-91.291,170.463,37.583,157.080
C03110=1044.260,135.705,-91.311,170.465,37.584,157.080
C03111=1044.267,135.954,-91.333,170.467,37.585,157.081
C03112=1044.272,136.202,-91.354,170.469,37.586,157.081
C03113=1044.279,136.451,-91.375,170.471,37.588,157.081
C03114=1044.285,136.700,-91.397,170.473,37.589,157.082
C03115=1044.290,136.949,-91.418,170.475,37.591,157.082
C03116=1044.297,137.199,-91.439,170.477,37.592,157.082
C03117=1044.303,137.448,-91.460,170.479,37.593,157.082
C03118=1044.310,137.697,-91.482,170.481,37.594,157.083
C03119=1044.315,137.945,-91.503,170.484,37.596,157.083
C03120=1044.321,138.194,-91.525,170.486,37.597,157.083
C03121=1044.328,138.443,-91.546,170.488,37.598,157.083
C03122=1044.334,138.692,-91.566,170.489,37.600,157.084
C03123=1044.340,138.942,-91.588,170.491,37.601,157.084
C03124=1044.346,139.191,-91.610,170.494,37.603,157.084
C03125=1044.353,139.440,-91.631,170.496,37.604,157.085
C03126=1044.358,139.688,-91.652,170.498,37.605,157.085
C03127=1044.364,139.938,-91.674,170.500,37.606,157.085
C03128=1044.371,140.187,-91.695,170.503,37.608,157.086
C03129=1044.376,140.435,-91.716,170.505,37.609,157.086
C03130=1044.382,140.684,-91.738,170.506,37.610,157.086
C03131=1044.389,140.934,-91.760,170.508,37.612,157.086
C03132=1044.395,141.219,-91.784,170.510,37.613,157.087
C03133=1044.403,141.505,-91.809,170.514,37.615,157.087
C03134=1044.409,141.790,-91.834,170.516,37.617,157.087
C03135=1044.416,142.076,-91.858,170.518,37.618,157.088
C03136=1044.422,142.326,-91.880,170.520,37.619,157.088
C03137=1044.428,142.575,-91.902,170.523,37.621,157.088
C03138=1044.434,142.823,-91.923,170.525,37.622,157.089
C03139=1044.440,143.072,-91.944,170.526,37.624,157.089
C03140=1044.446,143.322,-91.966,170.528,37.625,157.089
C03141=1044.453,143.571,-91.987,170.531,37.627,157.089
C03142=1044.459,143.818,-92.009,170.533,37.628,157.090
C03143=1044.465,144.068,-92.031,170.535,37.629,157.090
C03144=1044.471,144.317,-92.052,170.537,37.631,157.090
C03145=1044.478,144.566,-92.074,170.539,37.632,157.091
C03146=1044.484,144.815,-92.096,170.542,37.633,157.091
C03147=1044.489,145.064,-92.117,170.544,37.635,157.091
C03148=1044.496,145.313,-92.139,170.546,37.636,157.092
C03149=1044.502,145.562,-92.160,170.548,37.637,157.092
C03150=1044.508,145.811,-92.183,170.550,37.638,157.092
C03151=1044.514,146.060,-92.204,170.552,37.640,157.092
C03152=1044.520,146.309,-92.226,170.554,37.641,157.093
C03153=1044.527,146.558,-92.247,170.556,37.643,157.093
C03154=1044.532,146.807,-92.269,170.559,37.644,157.093
C03155=1044.538,147.056,-92.290,170.561,37.646,157.094
C03156=1044.545,147.305,-92.313,170.563,37.647,157.094
C03157=1044.551,147.554,-92.334,170.565,37.649,157.094
C03158=1044.557,147.803,-92.356,170.567,37.650,157.095
C03159=1044.563,148.052,-92.378,170.570,37.651,157.095
C03160=1044.570,148.301,-92.400,170.572,37.653,157.095
C03161=1044.575,148.549,-92.421,170.574,37.654,157.095
C03162=1044.581,148.799,-92.443,170.575,37.655,157.096
C03163=1044.587,149.047,-92.466,170.578,37.657,157.096
C03164=1044.593,149.297,-92.487,170.580,37.658,157.096
C03165=1044.600,149.546,-92.509,170.582,37.660,157.097
C03166=1044.606,149.794,-92.531,170.584,37.661,157.097
C03167=1044.612,150.044,-92.553,170.586,37.662,157.097
C03168=1044.617,150.292,-92.575,170.589,37.664,157.098
C03169=1044.624,150.541,-92.597,170.591,37.665,157.098
C03170=1044.630,150.790,-92.619,170.593,37.666,157.098
C03171=1044.636,151.039,-92.641,170.595,37.668,157.099
C03172=1044.642,151.288,-92.663,170.598,37.669,157.099
C03173=1044.648,151.538,-92.685,170.600,37.671,157.099
C03174=1044.654,151.786,-92.708,170.602,37.672,157.099
C03175=1044.660,152.035,-92.729,170.604,37.674,157.100
C03176=1044.667,152.285,-92.751,170.607,37.675,157.100
C03177=1044.672,152.533,-92.774,170.609,37.677,157.100
C03178=1044.678,152.783,-92.795,170.610,37.678,157.101
C03179=1044.684,153.031,-92.817,170.612,37.680,157.101
C03180=1044.690,153.280,-92.839,170.615,37.681,157.101
C03181=1044.697,153.528,-92.861,170.617,37.683,157.102
C03182=1044.702,153.778,-92.884,170.619,37.684,157.102
C03183=1044.709,154.026,-92.906,170.621,37.686,157.102
C03184=1044.715,154.276,-92.928,170.623,37.687,157.103
C03185=1044.721,154.524,-92.950,170.626,37.688,157.103
C03186=1044.727,154.774,-92.972,170.628,37.690,157.103
C03187=1044.733,155.022,-92.994,170.630,37.691,157.103
C03188=1044.739,155.272,-93.016,170.632,37.693,157.104
C03189=1044.745,155.520,-93.039,170.635,37.694,157.104
C03190=1044.751,155.770,-93.061,170.637,37.696,157.104
C03191=1044.757,156.019,-93.084,170.639,37.697,157.105
C03192=1044.764,156.267,-93.106,170.641,37.699,157.105
C03193=1044.770,156.516,-93.128,170.644,37.700,157.105
C03194=1044.775,156.765,-93.151,170.646,37.702,157.106
C03195=1044.782,157.014,-93.172,170.648,37.703,157.106
C03196=1044.789,157.299,-93.198,170.650,37.705,157.106
C03197=1044.796,157.585,-93.223,170.653,37.706,157.107
C03198=1044.803,157.870,-93.249,170.656,37.708,157.107
C03199=1044.809,158.155,-93.275,170.658,37.710,157.108
C03200=1044.815,158.404,-93.297,170.661,37.711,157.108
C03201=1044.822,158.652,-93.320,170.663,37.713,157.108
C03202=1044.827,158.902,-93.342,170.665,37.714,157.108
C03203=1044.834,159.151,-93.364,170.667,37.715,157.109
C03204=1044.840,159.400,-93.387,170.670,37.717,157.109
C03205=1044.846,159.649,-93.409,170.672,37.718,157.109
C03206=1044.853,159.898,-93.431,170.674,37.720,157.110
C03207=1044.859,160.147,-93.454,170.676,37.721,157.110
C03208=1044.865,160.395,-93.477,170.679,37.723,157.110
C03209=1044.870,160.645,-93.499,170.681,37.725,157.111
C03210=1044.876,160.894,-93.522,170.683,37.726,157.111
C03211=1044.883,161.142,-93.544,170.685,37.728,157.111
C03212=1044.888,161.391,-93.567,170.688,37.729,157.112
C03213=1044.894,161.640,-93.590,170.690,37.731,157.112
C03214=1044.900,161.889,-93.613,170.692,37.732,157.113
C03215=1044.905,162.139,-93.635,170.694,37.734,157.113
C03216=1044.912,162.387,-93.658,170.697,37.735,157.113
C03217=1044.917,162.636,-93.681,170.699,37.737,157.114
C03218=1044.923,162.885,-93.704,170.701,37.739,157.114
C03219=1044.929,163.134,-93.726,170.703,37.740,157.114
C03220=1044.935,163.382,-93.749,170.706,37.742,157.115
C03221=1044.941,163.631,-93.772,170.708,37.744,157.115
C03222=1044.947,163.880,-93.795,170.710,37.745,157.115
C03223=1044.953,164.129,-93.818,170.713,37.747,157.116
C03224=1044.958,164.378,-93.841,170.715,37.748,157.116
C03225=1044.965,164.627,-93.863,170.717,37.750,157.116
C03226=1044.971,164.876,-93.886,170.719,37.751,157.117
C03227=1044.976,165.124,-93.909,170.722,37.753,157.117
C03228=1044.982,165.373,-93.932,170.724,37.755,157.117
C03229=1044.988,165.622,-93.955,170.726,37.756,157.118
C03230=1044.995,165.872,-93.977,170.728,37.758,157.118
C03231=1045.001,166.120,-94.000,170.731,37.760,157.118
C03232=1045.006,166.369,-94.023,170.733,37.761,157.119
C03233=1045.012,166.618,-94.046,170.735,37.763,157.119
C03234=1045.018,166.867,-94.069,170.738,37.765,157.120
C03235=1045.023,167.116,-94.092,170.740,37.766,157.120
C03236=1045.030,167.365,-94.115,170.742,37.767,157.120
C03237=1045.036,167.613,-94.137,170.744,37.769,157.121
C03238=1045.042,167.862,-94.161,170.747,37.771,157.121
C03239=1045.048,168.111,-94.184,170.749,37.772,157.121
C03240=1045.054,168.360,-94.207,170.751,37.774,157.122
C03241=1045.060,168.609,-94.230,170.753,37.776,157.122
C03242=1045.066,168.858,-94.253,170.756,37.778,157.122
C03243=1045.072,169.107,-94.276,170.758,37.779,157.123
C03244=1045.077,169.356,-94.299,170.760,37.781,157.123
C03245=1045.084,169.605,-94.323,170.763,37.782,157.123
C03246=1045.090,169.853,-94.346,170.765,37.783,157.124
C03247=1045.096,170.102,-94.368,170.768,37.785,157.124
C03248=1045.102,170.351,-94.391,170.770,37.787,157.124
C03249=1045.108,170.600,-94.414,170.773,37.788,157.125
C03250=1045.114,170.848,-94.437,170.775,37.790,157.125
C03251=1045.120,171.098,-94.461,170.777,37.792,157.126
C03252=1045.126,171.347,-94.484,170.779,37.794,157.126
C03253=1045.132,171.595,-94.507,170.782,37.795,157.126
C03254=1045.138,171.843,-94.530,170.784,37.797,157.127
C03255=1045.145,172.093,-94.553,170.786,37.798,157.127
C03256=1045.150,172.342,-94.576,170.789,37.800,157.127
C03257=1045.156,172.591,-94.599,170.791,37.801,157.128
C03258=1045.162,172.839,-94.623,170.793,37.803,157.128
C03259=1045.168,173.089,-94.646,170.796,37.805,157.128
C03260=1045.175,173.373,-94.672,170.799,37.807,157.129
C03261=1045.182,173.658,-94.699,170.801,37.808,157.129
C03262=1045.190,173.943,-94.725,170.804,37.810,157.130
C03263=1045.196,174.227,-94.752,170.807,37.812,157.130
C03264=1045.203,174.477,-94.775,170.809,37.814,157.130
C03265=1045.208,174.726,-94.798,170.811,37.815,157.131
C03266=1045.214,174.974,-94.822,170.813,37.817,157.131
C03267=1045.220,175.223,-94.845,170.817,37.818,157.131
C03268=1045.227,175.472,-94.868,170.819,37.820,157.132
C03269=1045.233,175.721,-94.891,170.821,37.822,157.132
C03270=1045.239,175.969,-94.914,170.824,37.823,157.132
C03271=1045.246,176.218,-94.938,170.826,37.825,157.133
C03272=1045.251,176.467,-94.961,170.828,37.827,157.133
C03273=1045.257,176.716,-94.985,170.830,37.828,157.134
C03274=1045.264,176.965,-95.008,170.834,37.830,157.134
C03275=1045.269,177.214,-95.031,170.836,37.831,157.134
C03276=1045.276,177.463,-95.055,170.838,37.833,157.135
C03277=1045.283,177.712,-95.077,170.841,37.835,157.135
C03278=1045.289,177.960,-95.101,170.843,37.836,157.135
C03279=1045.295,178.210,-95.124,170.845,37.838,157.136
C03280=1045.301,178.458,-95.148,170.847,37.840,157.136
C03281=1045.307,178.707,-95.171,170.851,37.841,157.137
C03282=1045.313,178.956,-95.195,170.853,37.842,157.137
C03283=1045.319,179.204,-95.219,170.855,37.844,157.137
C03284=1045.326,179.454,-95.242,170.858,37.846,157.138
C03285=1045.332,179.702,-95.266,170.860,37.848,157.138
C03286=1045.337,179.951,-95.289,170.862,37.849,157.138
C03287=1045.344,180.200,-95.313,170.865,37.851,157.139
C03288=1045.350,180.449,-95.336,170.868,37.853,157.139
C03289=1045.357,180.697,-95.359,170.870,37.854,157.139
C03290=1045.363,180.946,-95.383,170.872,37.856,157.140
C03291=1045.370,181.195,-95.406,170.874,37.857,157.140
C03292=1045.376,181.443,-95.430,170.878,37.859,157.140
C03293=1045.382,181.693,-95.453,170.880,37.861,157.141
C03294=1045.388,181.941,-95.477,170.882,37.863,157.141
C03295=1045.395,182.190,-95.501,170.885,37.864,157.142
C03296=1045.400,182.439,-95.524,170.887,37.865,157.142
C03297=1045.407,182.688,-95.548,170.890,37.867,157.142
C03298=1045.413,182.936,-95.571,170.893,37.869,157.143
C03299=1045.419,183.186,-95.595,170.895,37.871,157.143
C03300=1045.425,183.434,-95.618,170.897,37.872,157.143
C03301=1045.432,183.683,-95.642,170.899,37.874,157.144
C03302=1045.438,183.932,-95.666,170.903,37.875,157.144
C03303=1045.445,184.181,-95.690,170.905,37.877,157.145
C03304=1045.450,184.430,-95.714,170.907,37.879,157.145
C03305=1045.456,184.678,-95.737,170.910,37.881,157.145
C03306=1045.462,184.927,-95.762,170.912,37.883,157.146
C03307=1045.468,185.176,-95.786,170.914,37.885,157.146
C03308=1045.474,185.425,-95.810,170.918,37.887,157.147
C03309=1045.480,185.673,-95.834,170.920,37.888,157.147
C03310=1045.485,185.922,-95.858,170.922,37.890,157.147
C03311=1045.492,186.171,-95.882,170.925,37.892,157.148
C03312=1045.497,186.419,-95.906,170.927,37.894,157.148
C03313=1045.504,186.668,-95.930,170.930,37.895,157.149
C03314=1045.509,186.917,-95.955,170.932,37.897,157.149
C03315=1045.515,187.166,-95.979,170.935,37.900,157.150
C03316=1045.521,187.414,-96.003,170.937,37.901,157.150
C03317=1045.527,187.663,-96.027,170.940,37.903,157.150
C03318=1045.533,187.912,-96.051,170.943,37.905,157.151
C03319=1045.539,188.161,-96.075,170.945,37.907,157.151
C03320=1045.545,188.410,-96.099,170.947,37.908,157.151
C03321=1045.551,188.659,-96.123,170.950,37.910,157.152
C03322=1045.557,188.907,-96.148,170.952,37.912,157.152
C03323=1045.563,189.156,-96.172,170.955,37.914,157.153
C03324=1045.570,189.440,-96.199,170.958,37.916,157.153
C03325=1045.577,189.724,-96.227,170.961,37.918,157.154
C03326=1045.583,190.010,-96.255,170.964,37.920,157.154
C03327=1045.591,190.294,-96.283,170.967,37.923,157.155
C03328=1045.597,190.542,-96.307,170.969,37.924,157.155
C03329=1045.603,190.791,-96.331,170.972,37.926,157.155
C03330=1045.609,191.040,-96.355,170.974,37.928,157.156
C03331=1045.615,191.289,-96.379,170.977,37.930,157.156
C03332=1045.620,191.538,-96.404,170.980,37.932,157.157
C03333=1045.626,191.787,-96.428,170.982,37.934,157.157
C03334=1045.632,192.035,-96.453,170.984,37.935,157.158
C03335=1045.639,192.283,-96.477,170.988,37.937,157.158
C03336=1045.645,192.533,-96.501,170.990,37.939,157.158
C03337=1045.651,192.781,-96.525,170.992,37.941,157.159
C03338=1045.657,193.030,-96.550,170.996,37.943,157.159
C03339=1045.664,193.279,-96.574,170.998,37.945,157.160
C03340=1045.669,193.527,-96.599,171.000,37.947,157.160
C03341=1045.675,193.776,-96.623,171.003,37.948,157.160
C03342=1045.681,194.024,-96.648,171.006,37.950,157.161
C03343=1045.688,194.273,-96.672,171.008,37.952,157.161
C03344=1045.694,194.523,-96.696,171.011,37.954,157.162
C03345=1045.699,194.771,-96.721,171.014,37.956,157.162
C03346=1045.706,195.019,-96.745,171.016,37.958,157.163
C03347=1045.712,195.269,-96.770,171.019,37.959,157.163
C03348=1045.718,195.517,-96.794,171.021,37.962,157.163
C03349=1045.724,195.766,-96.819,171.024,37.964,157.164
C03350=1045.731,196.015,-96.843,171.027,37.965,157.164
C03351=1045.736,196.263,-96.867,171.029,37.967,157.165
C03352=1045.743,196.512,-96.892,171.032,37.969,157.165
C03353=1045.749,196.761,-96.917,171.035,37.971,157.166
C03354=1045.755,197.010,-96.942,171.037,37.973,157.166
C03355=1045.761,197.258,-96.966,171.040,37.975,157.166
C03356=1045.767,197.507,-96.990,171.043,37.976,157.167
C03357=1045.774,197.755,-97.015,171.045,37.979,157.167
C03358=1045.780,198.005,-97.040,171.048,37.981,157.168
C03359=1045.786,198.252,-97.064,171.051,37.982,157.168
C03360=1045.792,198.502,-97.089,171.053,37.984,157.169
C03361=1045.798,198.750,-97.114,171.056,37.986,157.169
C03362=1045.805,198.999,-97.138,171.059,37.988,157.169
C03363=1045.810,199.247,-97.163,171.061,37.990,157.170
C03364=1045.817,199.496,-97.187,171.064,37.992,157.170
C03365=1045.823,199.745,-97.212,171.067,37.994,157.171
C03366=1045.829,199.994,-97.237,171.069,37.996,157.171
C03367=1045.836,200.243,-97.262,171.072,37.997,157.172
C03368=1045.841,200.491,-97.286,171.075,37.999,157.172
C03369=1045.848,200.740,-97.311,171.077,38.002,157.172
C03370=1045.854,200.989,-97.335,171.080,38.003,157.173
C03371=1045.860,201.238,-97.361,171.083,38.005,157.173
C03372=1045.867,201.486,-97.385,171.085,38.007,157.174
C03373=1045.873,201.734,-97.410,171.089,38.009,157.174
C03374=1045.879,201.983,-97.435,171.091,38.011,157.175
C03375=1045.885,202.232,-97.460,171.094,38.013,157.175
C03376=1045.891,202.481,-97.485,171.097,38.015,157.176
C03377=1045.897,202.730,-97.510,171.099,38.017,157.176
C03378=1045.903,202.978,-97.535,171.102,38.019,157.176
C03379=1045.909,203.227,-97.560,171.105,38.021,157.177
C03380=1045.915,203.476,-97.585,171.107,38.023,157.177
C03381=1045.921,203.724,-97.610,171.110,38.026,157.178
C03382=1045.927,203.973,-97.636,171.113,38.027,157.178
C03383=1045.933,204.222,-97.660,171.115,38.030,157.179
C03384=1045.940,204.470,-97.685,171.119,38.031,157.179
C03385=1045.946,204.719,-97.710,171.121,38.034,157.180
C03386=1045.952,204.967,-97.735,171.124,38.035,157.180
C03387=1045.958,205.216,-97.761,171.127,38.038,157.181
C03388=1045.983,206.268,-97.868,171.381,38.138,157.206
C03389=1045.991,206.543,-97.896,171.382,38.141,157.206
C03390=1045.998,206.817,-97.925,171.385,38.144,157.207
C03391=1046.006,207.092,-97.954,171.387,38.147,157.208
C03392=1046.013,207.367,-97.983,171.389,38.151,157.209
C03393=1046.020,207.616,-98.009,171.392,38.153,157.209
C03394=1046.026,207.864,-98.035,171.393,38.156,157.210
C03395=1046.033,208.113,-98.062,171.396,38.159,157.210
C03396=1046.039,208.361,-98.088,171.398,38.162,157.211
C03397=1046.046,208.610,-98.115,171.400,38.164,157.212
C03398=1046.052,208.858,-98.142,171.402,38.167,157.212
C03399=1046.058,209.107,-98.167,171.404,38.170,157.213
C03400=1046.065,209.355,-98.193,171.406,38.173,157.214
C03401=1046.071,209.604,-98.220,171.408,38.175,157.214
C03402=1046.078,209.852,-98.246,171.410,38.178,157.215
C03403=1046.085,210.101,-98.272,171.413,38.181,157.215
C03404=1046.091,210.350,-98.299,171.414,38.184,157.216
C03405=1046.098,210.598,-98.325,171.417,38.187,157.217
C03406=1046.105,210.846,-98.352,171.418,38.190,157.217
C03407=1046.111,211.095,-98.379,171.421,38.193,157.218
C03408=1046.118,211.343,-98.405,171.422,38.196,157.219
C03409=1046.123,211.592,-98.432,171.425,38.198,157.219
C03410=1046.131,211.841,-98.458,171.427,38.201,157.220
C03411=1046.137,212.089,-98.486,171.429,38.204,157.220
C03412=1046.144,212.337,-98.512,171.431,38.207,157.221
C03413=1046.150,212.586,-98.539,171.433,38.209,157.222
C03414=1046.157,212.834,-98.565,171.435,38.212,157.222
C03415=1046.163,213.083,-98.592,171.438,38.215,157.223
C03416=1046.170,213.331,-98.618,171.440,38.218,157.224
C03417=1046.176,213.580,-98.645,171.442,38.220,157.224
C03418=1046.182,213.828,-98.671,171.444,38.223,157.225
C03419=1046.189,214.077,-98.699,171.446,38.226,157.225
C03420=1046.196,214.325,-98.725,171.449,38.229,157.226
C03421=1046.202,214.574,-98.752,171.450,38.232,157.227
C03422=1046.208,214.822,-98.778,171.453,38.235,157.227
C03423=1046.215,215.071,-98.805,171.454,38.238,157.228
C03424=1046.221,215.319,-98.832,171.457,38.241,157.229
C03425=1046.228,215.568,-98.859,171.459,38.243,157.229
C03426=1046.234,215.817,-98.886,171.461,38.246,157.230
C03427=1046.241,216.065,-98.912,171.463,38.249,157.230
C03428=1046.248,216.313,-98.939,171.466,38.252,157.231
C03429=1046.253,216.561,-98.966,171.467,38.254,157.232
C03430=1046.261,216.810,-98.993,171.470,38.257,157.232
C03431=1046.267,217.059,-99.020,171.472,38.260,157.233
C03432=1046.274,217.307,-99.046,171.474,38.262,157.233
C03433=1046.280,217.556,-99.073,171.476,38.265,157.234
C03434=1046.286,217.805,-99.100,171.479,38.268,157.235
C03435=1046.293,218.052,-99.127,171.480,38.271,157.235
C03436=1046.300,218.301,-99.154,171.483,38.274,157.236
C03437=1046.306,218.549,-99.180,171.485,38.277,157.237
C03438=1046.313,218.798,-99.208,171.487,38.280,157.237
C03439=1046.319,219.047,-99.235,171.489,38.282,157.238
C03440=1046.326,219.294,-99.262,171.492,38.285,157.239
C03441=1046.332,219.543,-99.289,171.494,38.288,157.239
C03442=1046.340,219.792,-99.315,171.496,38.290,157.240
C03443=1046.346,220.041,-99.343,171.499,38.293,157.240
C03444=1046.352,220.289,-99.370,171.500,38.296,157.241
C03445=1046.359,220.569,-99.400,171.503,38.299,157.242
C03446=1046.367,220.849,-99.431,171.505,38.302,157.242
C03447=1046.375,221.129,-99.461,171.508,38.305,157.243
C03448=1046.381,221.410,-99.492,171.511,38.308,157.244
C03449=1046.388,221.658,-99.519,171.513,38.311,157.244
C03450=1046.395,221.907,-99.546,171.515,38.314,157.245
C03451=1046.401,222.155,-99.573,171.517,38.317,157.246
C03452=1046.407,222.404,-99.600,171.520,38.320,157.246
C03453=1046.414,222.652,-99.628,171.522,38.323,157.247
C03454=1046.420,222.900,-99.655,171.524,38.325,157.248
C03455=1046.427,223.149,-99.682,171.526,38.328,157.248
C03456=1046.433,223.397,-99.710,171.529,38.331,157.249
C03457=1046.440,223.646,-99.736,171.530,38.334,157.250
C03458=1046.446,223.894,-99.764,171.533,38.336,157.250
C03459=1046.453,224.142,-99.792,171.535,38.339,157.251
C03460=1046.459,224.391,-99.819,171.538,38.342,157.251
C03461=1046.466,224.639,-99.846,171.539,38.344,157.252
C03462=1046.472,224.888,-99.874,171.542,38.347,157.253
C03463=1046.479,225.137,-99.901,171.545,38.350,157.253
C03464=1046.485,225.385,-99.928,171.547,38.353,157.254
C03465=1046.492,225.633,-99.955,171.549,38.355,157.254
C03466=1046.498,225.882,-99.982,171.551,38.358,157.255
C03467=1046.505,226.130,-100.010,171.554,38.361,157.256
C03468=1046.512,226.379,-100.038,171.556,38.364,157.256
C03469=1046.518,226.628,-100.065,171.558,38.367,157.257
C03470=1046.524,226.875,-100.092,171.560,38.370,157.258
C03471=1046.531,227.124,-100.120,171.563,38.372,157.258
C03472=1046.538,227.372,-100.147,171.565,38.375,157.259
C03473=1046.544,227.621,-100.174,171.567,38.378,157.260
C03474=1046.551,227.869,-100.202,171.569,38.380,157.260
C03475=1046.558,228.117,-100.229,171.572,38.383,157.261
C03476=1046.564,228.366,-100.257,171.574,38.386,157.261
C03477=1046.571,228.614,-100.284,171.577,38.388,157.262
C03478=1046.577,228.863,-100.311,171.578,38.391,157.263
C03479=1046.584,229.112,-100.339,171.581,38.394,157.263
C03480=1046.590,229.359,-100.367,171.584,38.396,157.264
C03481=1046.597,229.608,-100.394,171.586,38.399,157.264
C03482=1046.603,229.856,-100.423,171.589,38.402,157.265
C03483=1046.609,230.105,-100.450,171.590,38.405,157.266
C03484=1046.616,230.353,-100.478,171.593,38.408,157.266
C03485=1046.623,230.602,-100.506,171.595,38.411,157.267
C03486=1046.629,230.849,-100.533,171.598,38.413,157.268
C03487=1046.635,231.098,-100.561,171.600,38.416,157.268
C03488=1046.642,231.346,-100.589,171.602,38.419,157.269
C03489=1046.649,231.595,-100.616,171.604,38.422,157.270
C03490=1046.655,231.844,-100.645,171.607,38.424,157.270
C03491=1046.661,232.092,-100.672,171.609,38.427,157.271
C03492=1046.668,232.340,-100.700,171.612,38.430,157.271
C03493=1046.674,232.588,-100.727,171.614,38.433,157.272
C03494=1046.681,232.837,-100.755,171.616,38.435,157.273
C03495=1046.687,233.085,-100.784,171.619,38.438,157.273
C03496=1046.694,233.334,-100.811,171.621,38.441,157.274
C03497=1046.700,233.582,-100.839,171.624,38.444,157.275
C03498=1046.707,233.831,-100.867,171.626,38.446,157.275
C03499=1046.713,234.079,-100.895,171.628,38.449,157.276
C03500=1046.720,234.328,-100.923,171.630,38.452,157.277
C03501=1046.726,234.600,-100.953,171.633,38.455,157.277
C03502=1046.734,234.873,-100.984,171.636,38.458,157.278
C03503=1046.741,235.145,-101.014,171.638,38.461,157.279
C03504=1046.748,235.418,-101.046,171.641,38.464,157.279
C03505=1046.754,235.666,-101.074,171.643,38.467,157.280
C03506=1046.761,235.915,-101.102,171.646,38.470,157.281
C03507=1046.768,236.163,-101.130,171.649,38.472,157.281
C03508=1046.774,236.412,-101.157,171.651,38.475,157.282
C03509=1046.781,236.660,-101.186,171.654,38.478,157.282
C03510=1046.787,236.908,-101.214,171.656,38.481,157.283
C03511=1046.794,237.157,-101.242,171.659,38.484,157.284
C03512=1046.800,237.406,-101.270,171.660,38.486,157.284
C03513=1046.807,237.653,-101.299,171.663,38.489,157.285
C03514=1046.813,237.902,-101.326,171.665,38.492,157.286
C03515=1046.820,238.150,-101.354,171.668,38.494,157.286
C03516=1046.826,238.399,-101.382,171.670,38.497,157.287
C03517=1046.833,238.647,-101.411,171.673,38.500,157.288
C03518=1046.840,238.895,-101.439,171.675,38.502,157.288
C03519=1046.846,239.144,-101.467,171.678,38.505,157.289
C03520=1046.853,239.392,-101.495,171.681,38.508,157.289
C03521=1046.859,239.641,-101.524,171.683,38.510,157.290
C03522=1046.866,239.888,-101.552,171.686,38.513,157.291
C03523=1046.872,240.137,-101.580,171.687,38.516,157.291
C03524=1046.878,240.386,-101.608,171.690,38.519,157.292
C03525=1046.885,240.633,-101.637,171.692,38.521,157.293
C03526=1046.892,240.882,-101.664,171.695,38.524,157.293
C03527=1046.898,241.130,-101.693,171.697,38.527,157.294
C03528=1046.905,241.378,-101.721,171.700,38.529,157.294
C03529=1046.911,241.627,-101.750,171.703,38.532,157.295
C03530=1046.918,241.875,-101.778,171.705,38.535,157.296
C03531=1046.924,242.123,-101.807,171.708,38.538,157.297
C03532=1046.931,242.372,-101.835,171.710,38.541,157.297
C03533=1046.937,242.620,-101.864,171.713,38.543,157.298
C03534=1046.943,242.868,-101.892,171.715,38.546,157.298
C03535=1046.950,243.116,-101.920,171.718,38.549,157.299
C03536=1046.956,243.365,-101.949,171.720,38.552,157.300
C03537=1046.963,243.613,-101.977,171.723,38.554,157.300
C03538=1046.969,243.861,-102.006,171.726,38.557,157.301
C03539=1046.975,244.110,-102.035,171.728,38.560,157.302
C03540=1046.982,244.358,-102.063,171.731,38.563,157.302
C03541=1046.988,244.606,-102.092,171.732,38.565,157.303
C03542=1046.996,244.855,-102.120,171.735,38.568,157.304
C03543=1047.002,245.103,-102.149,171.737,38.571,157.304
C03544=1047.008,245.351,-102.178,171.740,38.574,157.305
C03545=1047.015,245.600,-102.206,171.743,38.576,157.305
C03546=1047.021,245.848,-102.235,171.745,38.579,157.306
C03547=1047.027,246.096,-102.264,171.748,38.582,157.307
C03548=1047.033,246.345,-102.292,171.750,38.585,157.307
C03549=1047.039,246.593,-102.321,171.753,38.588,157.308
C03550=1047.046,246.841,-102.350,171.755,38.591,157.309
C03551=1047.053,247.089,-102.379,171.758,38.593,157.309
C03552=1047.059,247.337,-102.408,171.761,38.596,157.310
C03553=1047.066,247.586,-102.437,171.763,38.599,157.311
C03554=1047.072,247.834,-102.466,171.766,38.602,157.311
C03555=1047.078,248.083,-102.495,171.768,38.605,157.312
C03556=1047.084,248.331,-102.524,171.771,38.608,157.313
C03557=1047.091,248.597,-102.554,171.774,38.611,157.313
C03558=1047.098,248.864,-102.586,171.776,38.614,157.314
C03559=1047.105,249.131,-102.617,171.780,38.616,157.315
C03560=1047.112,249.398,-102.649,171.782,38.619,157.316
C03561=1047.119,249.646,-102.677,171.785,38.622,157.316
C03562=1047.125,249.894,-102.706,171.788,38.625,157.317
C03563=1047.131,250.143,-102.734,171.790,38.628,157.318
C03564=1047.137,250.391,-102.763,171.793,38.631,157.318
C03565=1047.144,250.640,-102.793,171.795,38.633,157.319
C03566=1047.150,250.888,-102.822,171.798,38.636,157.319
C03567=1047.156,251.136,-102.851,171.800,38.639,157.320
C03568=1047.163,251.384,-102.880,171.803,38.642,157.321
C03569=1047.169,251.632,-102.909,171.806,38.645,157.321
C03570=1047.177,251.881,-102.938,171.808,38.648,157.322
C03571=1047.183,252.129,-102.967,171.811,38.650,157.323
C03572=1047.189,252.376,-102.997,171.813,38.653,157.323
C03573=1047.196,252.625,-103.026,171.816,38.656,157.324
C03574=1047.202,252.873,-103.055,171.819,38.659,157.325
C03575=1047.209,253.122,-103.084,171.822,38.661,157.325
C03576=1047.215,253.370,-103.113,171.825,38.664,157.326
C03577=1047.221,253.618,-103.142,171.827,38.667,157.327
C03578=1047.228,253.867,-103.172,171.830,38.669,157.327
C03579=1047.234,254.115,-103.201,171.832,38.672,157.328
C03580=1047.241,254.363,-103.229,171.835,38.675,157.329
C03581=1047.248,254.610,-103.259,171.838,38.678,157.329
C03582=1047.255,254.859,-103.288,171.840,38.680,157.330
C03583=1047.261,255.107,-103.317,171.843,38.683,157.331
C03584=1047.267,255.355,-103.346,171.845,38.686,157.331
C03585=1047.274,255.604,-103.376,171.848,38.689,157.332
C03586=1047.280,255.852,-103.405,171.851,38.691,157.333
C03587=1047.287,256.100,-103.435,171.854,38.694,157.333
C03588=1047.294,256.349,-103.464,171.857,38.697,157.334
C03589=1047.300,256.597,-103.493,171.859,38.700,157.335
C03590=1047.306,256.845,-103.522,171.862,38.702,157.335
C03591=1047.313,257.093,-103.552,171.864,38.705,157.336
C03592=1047.320,257.341,-103.581,171.867,38.708,157.337
C03593=1047.326,257.589,-103.610,171.871,38.711,157.337
C03594=1047.333,257.837,-103.640,171.873,38.714,157.338
C03595=1047.340,258.085,-103.669,171.876,38.716,157.338
C03596=1047.347,258.334,-103.698,171.878,38.719,157.339
C03597=1047.353,258.582,-103.728,171.881,38.722,157.340
C03598=1047.360,258.830,-103.757,171.884,38.725,157.341
C03599=1047.366,259.079,-103.786,171.887,38.727,157.341
C03600=1047.373,259.326,-103.816,171.890,38.730,157.342
C03601=1047.380,259.575,-103.846,171.892,38.733,157.342
C03602=1047.386,259.822,-103.875,171.895,38.736,157.343
C03603=1047.393,260.071,-103.905,171.897,38.738,157.344
C03604=1047.400,260.319,-103.934,171.900,38.741,157.344
C03605=1047.406,260.567,-103.964,171.904,38.743,157.345
C03606=1047.413,260.816,-103.993,171.906,38.746,157.346
C03607=1047.420,261.063,-104.023,171.909,38.749,157.346
C03608=1047.426,261.312,-104.052,171.911,38.752,157.347
C03609=1047.433,261.560,-104.082,171.914,38.754,157.348
C03610=1047.440,261.808,-104.111,171.918,38.757,157.348
C03611=1047.446,262.056,-104.141,171.920,38.760,157.349
C03612=1047.453,262.305,-104.170,171.923,38.762,157.350
C03613=1047.461,262.570,-104.202,171.925,38.765,157.350
C03614=1047.467,262.835,-104.234,171.929,38.769,157.351
C03615=1047.474,263.101,-104.266,171.932,38.772,157.352
C03616=1047.481,263.366,-104.298,171.935,38.774,157.353
C03617=1047.487,263.614,-104.328,171.938,38.777,157.353
C03618=1047.494,263.863,-104.358,171.940,38.780,157.354
C03619=1047.501,264.110,-104.387,171.943,38.783,157.355
C03620=1047.507,264.359,-104.418,171.946,38.786,157.355
C03621=1047.513,264.607,-104.447,171.949,38.789,157.356
C03622=1047.520,264.854,-104.477,171.952,38.792,157.357
C03623=1047.526,265.103,-104.508,171.955,38.794,157.357
